	sEcSlaveAmsNetAdr:T_AmsNetId;
	rValue:REAL;
	bOverrange, bDataInvalid, bError, bCalibrationInProgress, bSteadyState:BOOL;
	bTxPDOToggle, bSyncError:BOOL;
	sfFullCalibration:R_TRIG;
	sfZeroCalibration:R_TRIG;
	sfTara:R_TRIG;
	sfTaraEEProm:R_TRIG;
	fbCoE:FB_EcCoESdoWrite;
	wCoeData:WORD;
	sStatus, sSampleMode:STRING(100);
	bTermError:BOOL;
	nCntCalibrations:UDINT;
	sfCalibInProgress:R_TRIG;
	sfLoadReference:R_TRIG;
	sfScaleFactor:R_TRIG;
	rValueDiff, rValueL:REAL;
	bActivateAutoInputFreeze:BOOL;
	rInputFreezeTreshold:REAL:=10;
	tofInputFreeze:TOF;
	tInputFreeze:TIME:=t#50ms;
	sfCntInputFreeze:R_TRIG;
	nCntInputFreeze:UDINT;
	rScaleFactor :REAL:=1.0;
	bCmdScaleFactor:BOOL;


END_VAR

(*EP3356-0022)	para celdas de carga*)
(*toma de datos*)
bOverrange		:= wStatus.1;
bDataInvalid	:= wStatus.3;
bError			:= wStatus.6;
bCalibrationInProgress := wStatus.7;
bSteadyState	:= wStatus.8;
bSyncError		:= wStatus.13;
bTxPDOToggle	:= wStatus.15;

(*triggers*)
sfScaleFactor(CLK:=bCmdScaleFactor);
sfZeroCalibration(CLK:=bCmd_ZeroCalibration);
sfFullCalibration(CLK:=bCmd_FullCalibration);
sfTara(CLK:=bCmd_Tara);
sfTaraEEProm(CLK:=bCmd_TaraEEProm);
sfLoadReference(CLK:=bCmd_LoadReference);

(*value: Integer or Real value*)
IF (rValue_REAL <> 0) THEN	(*select currently used input data*)
	rValue := rValue_REAL;
ELSIF (nValue_DINT <> 0) THEN
	rValue := DINT_TO_REAL(nValue_DINT)/1000;
ELSE
	rValue := 0;
END_IF

(*status*)
IF bWcState THEN
	sStatus := 'Wc fail';
	bTermError := TRUE;
ELSIF NOT (wState.3) THEN
	sStatus := 'Slave not in OP';
	bTermError := TRUE;
ELSIF bDataInvalid THEN
	sStatus := 'DataInvalid';
	bTermError := TRUE;
ELSIF bError THEN
	sStatus := 'Channel Error';
	bTermError := TRUE;
ELSIF bOverrange THEN
	sStatus := 'Overrange';
	bTermError := TRUE;
ELSE
	sStatus := 'ok';
	bTermError := FALSE;
END_IF

	(*sample mode 0/1*)
sSampleMode := SEL(bSampleMode, '0', '1');

	(*count calibrations*)
sfCalibInProgress(CLK:= bCalibrationInProgress, Q=> );
nCntCalibrations := SEL(sfCalibInProgress.Q , nCntCalibrations, nCntCalibrations+ 1);

	(*Coe parameter administration*)
sEcSlaveAmsNetAdr := F_CreateAmsNetId(nIds:=stEcSlaveAmsNetAdr.netId );

	(*test input freeze
this lines are for a small demonstration of Input freeze: when difference of loadvalue, compared to last PLC cycle, is over rInputFreezeTreshold
then InputFreeze is activated by tofInputFreeze for some time. See screenshot in documentation for further explanations*)
rValueDiff := rValue - rValueL;
rValueL := rValue;
tofInputFreeze(IN:= bActivateAutoInputFreeze AND (ABS(rValueDiff) >rInputFreezeTreshold) , PT:= tInputFreeze, Q=> , ET=> );
sfCntInputFreeze(CLK:= tofInputFreeze.Q , Q=> );
nCntInputFreeze := SEL(sfCntInputFreeze.Q , nCntInputFreeze, nCntInputFreeze+ 1);

(*++++++++++++++ comunicacion CoE  ++++++++++++++++++++++*)
(* Scale factor*)
fbCoE(
	sNetId		:= sEcSlaveAmsNetAdr,
	nSlaveAddr 	:= stEcSlaveAmsNetAdr.port,
	nSubIndex 	:= 16#27,
	nIndex 		:= 16#8000,
	pSrcBuf 	:= ADR(rScaleFactor),
	cbBufLen 	:= SIZEOF(rScaleFactor),
	bExecute 	:= sfScaleFactor.Q,
	tTimeout 	:= t#5s
);

wCoeData := 16#0101; (* Comando zerocalibration*)
fbCoE(
	sNetId		:= sEcSlaveAmsNetAdr,
	nSlaveAddr 	:= stEcSlaveAmsNetAdr.port,
	nSubIndex 	:= 16#01,
	nIndex 		:= 16#FB00,
	pSrcBuf 	:= ADR(wCoeData),
	cbBufLen 	:= SIZEOF(wCoeData),
	bExecute 	:= sfZeroCalibration.Q,
	tTimeout 	:= t#5s
);

wCoeData := 16#0102; (* calibracion*)
fbCoE(
	sNetId		:= sEcSlaveAmsNetAdr,
	nSlaveAddr 	:= stEcSlaveAmsNetAdr.port,
	nSubIndex 	:= 16#01,
	nIndex 		:= 16#FB00,
	pSrcBuf 	:= ADR(wCoeData),
	cbBufLen 	:= SIZEOF(wCoeData),
	bExecute 	:= sfFullCalibration.Q,
	tTimeout 	:= t#5s
);

wCoeData := 16#0001; (* tara*)
fbCoE(
	sNetId		:= sEcSlaveAmsNetAdr,
	nSlaveAddr 	:= stEcSlaveAmsNetAdr.port,
	nSubIndex 	:= 16#01,
	nIndex 		:= 16#FB00,
	pSrcBuf 	:= ADR(wCoeData),
	cbBufLen 	:= SIZEOF(wCoeData),
	bExecute 	:= sfTara.Q,
	tTimeout 	:= t#5s
);

wCoeData := 16#0002; (* tara EEProm*)
fbCoE(
	sNetId		:= sEcSlaveAmsNetAdr,
	nSlaveAddr 	:= stEcSlaveAmsNetAdr.port,
	nSubIndex 	:= 16#01,
	nIndex 		:= 16#FB00,
	pSrcBuf 	:= ADR(wCoeData),
	cbBufLen 	:= SIZEOF(wCoeData),
	bExecute 	:= sfTaraEEProm.Q,
	tTimeout 	:= t#5s
);

(* load reference*)
fbCoE(
	sNetId		:= sEcSlaveAmsNetAdr,
	nSlaveAddr 	:= stEcSlaveAmsNetAdr.port,
	nSubIndex 	:= 16#28,
	nIndex 		:= 16#8000,
	pSrcBuf 	:= ADR(fLoadReference),
	cbBufLen 	:= SIZEOF(fLoadReference),
	bExecute 	:= sfLoadReference.Q,
	tTimeout 	:= t#5s
);


	(*output data to terminal*)
wControl.0 := bStartManualCalib;
wControl.1 := bDisableCalibration;
wControl.2 := bInputFreeze OR tofInputFreeze.Q ;
wControl.3 := bSampleMode;
wControl.4 := bTara;

END_FUNCTION_BLOCK

// ---- POUs/Tabla_FIFO.TcPOU
FUNCTION_BLOCK Tabla_FIFO
VAR_INPUT 
	Dato :REAL;
END_VAR
VAR_OUTPUT
END_VAR
VAR_IN_OUT
	Tabla :ARRAY [1..10]OF REAL;
	Trigger :BOOL;
END_VAR
VAR
	posicion: INT;
END_VAR

IF trigger  THEN
	posicion:=1;
	FOR posicion:=10 TO 2 BY -1 DO
	Tabla[posicion]:=Tabla[posicion-1];
	END_FOR;
	Tabla[1]:=Dato;
	trigger:=FALSE;
END_IF

END_FUNCTION_BLOCK

// ---- POUs/Perifericos/Descarga_semilla.TcPOU
PROGRAM Descarga_semilla
VAR
	fbPE_B_VF1 :Equipo_Motor_ATV320;//Elevador embolse
	PE_B1_V1: Equipo_Valvula_5_2_biestable;
	PE_B1_V1_CmdAuto_Pos1:BOOL;
	PE_B1_V1_CmdAuto_Pos2:BOOL;
	PE_B2_V1: Equipo_Valvula_5_2_biestable;
	PE_B2_V1_CmdAuto_Pos1:BOOL;
	PE_B2_V1_CmdAuto_Pos2:BOOL;
	PE_B3_V1: Equipo_Valvula_5_2_biestable;
	PE_B3_V1_CmdAuto_Pos1:BOOL;
	PE_B3_V1_CmdAuto_Pos2:BOOL;
	PE_B1_V2_CmdAuto:BOOL;
	PE_B2_V2_CmdAuto:BOOL;
	PE_B3_V2_CmdAuto:BOOL;	
	
	bHS :BOOL;
	dintHS	:DINT:=3;
	Tmr_B1_LLS: TON;
	B1_LLS_Ok: BOOL;
	Tmr_B2_LLS: TON;
	B2_LLS_Ok: BOOL;
	TmrCicloCarga: TON;
	Cargar_B2: BOOL;
	AuxCargar_B2: BOOL;
	AuxB1_V1: BOOL;
	AuxB2_V1: BOOL;
	TmrDemoraB2_V1: TOF;
	TmrPE_B1_HLS: TON;	//Nível alto da caixa de sacarias
	TmrPE_B2_HLS: TON;	//Nível alto do BIGBAG 2
	TmrPE_B3_HLS: TON;	//Nível alto do BIGBAG 3
	TDemoraPE_B1_LLS: TON;
	TDemoraPE_BE2_LLS: TON;
	TDemoraPE_BE3_LLS: TON;
	Tmr_B3_LLS: TON;
	B3_LLS_Ok: BOOL;
	Tiempo_seg_to_TIME_PE_B_VF1: Tiempo_seg_to_TIME;
	TmrDemoraPE_B_VF1: TOF;
	TDemoraB3_V1: TOF;
	PE_B1_V1_Teste: Equipo_Valvula_5_2;
	PE_B1_V2_Teste: Equipo_Valvula_5_2;
	PE_B1_V3_Teste: Equipo_Valvula_5_2;
	TON_CaixaCheia: TON;
	PausaEnsaque: BOOL;	//Se as duas caixas de ensaque estiverem cheias e a descarga for no bigbag, pausa o processo
	// Atraso na descarga da caixa 3 para que não passem canecas cheias
	TOF_DescargaCX3: TOF;
END_VAR
VAR // added by the converter: edge detectors and wires of the graphical bodies
    _w1 : BOOL;
    _rt1 : R_TRIG;
END_VAR

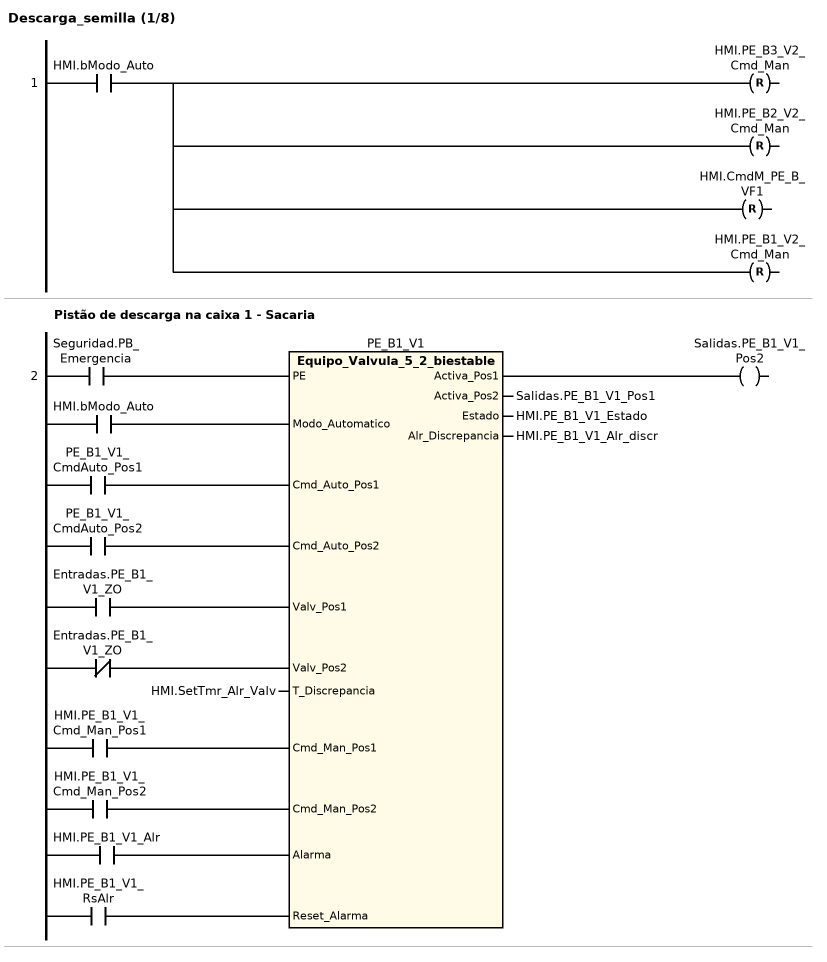
// NETWORK 1
_w1 := HMI.bModo_Auto;
HMI.PE_B3_V2_Cmd_Man R= _w1;
HMI.PE_B2_V2_Cmd_Man R= _w1;
HMI.CmdM_PE_B_VF1 R= _w1;
HMI.PE_B1_V2_Cmd_Man R= _w1;

// NETWORK 2: Pistão de descarga na caixa 1 - Sacaria
PE_B1_V1(
    PE := Seguridad.PB_Emergencia,
    Modo_Automatico := HMI.bModo_Auto,
    Cmd_Auto_Pos1 := PE_B1_V1_CmdAuto_Pos1,
    Cmd_Auto_Pos2 := PE_B1_V1_CmdAuto_Pos2,
    Valv_Pos1 := Entradas.PE_B1_V1_ZO,
    Valv_Pos2 := NOT Entradas.PE_B1_V1_ZO,
    T_Discrepancia := HMI.SetTmr_Alr_Valv,
    Cmd_Man_Pos1 := HMI.PE_B1_V1_Cmd_Man_Pos1,
    Cmd_Man_Pos2 := HMI.PE_B1_V1_Cmd_Man_Pos2,
    Alarma := HMI.PE_B1_V1_Alr,
    Reset_Alarma := HMI.PE_B1_V1_RsAlr,
    Activa_Pos2 => Salidas.PE_B1_V1_Pos1,
    Estado => HMI.PE_B1_V1_Estado,
    Alr_Discrepancia => HMI.PE_B1_V1_Alr_discr); // Equipo_Valvula_5_2_biestable
Salidas.PE_B1_V1_Pos2 := PE_B1_V1.Activa_Pos1;

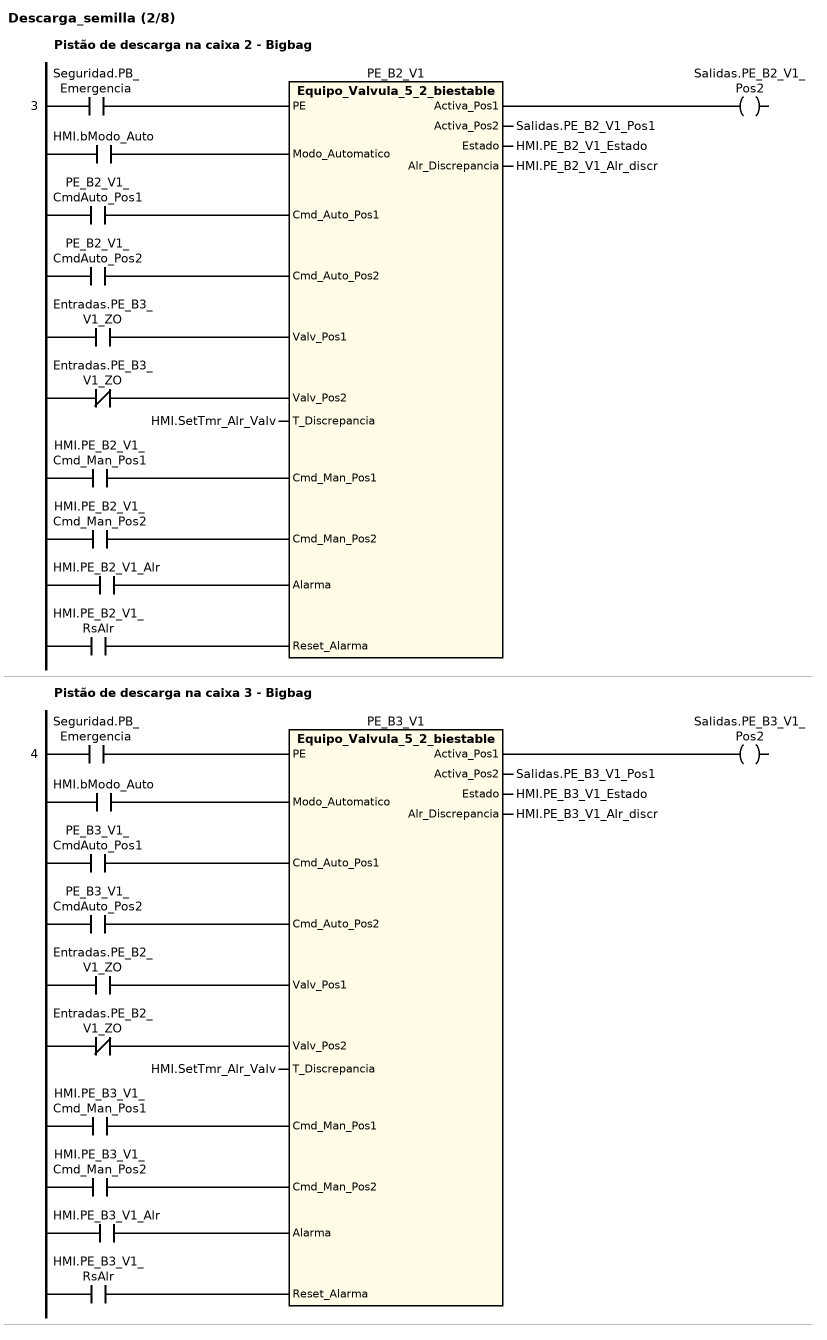
// NETWORK 3: Pistão de descarga na caixa 2 - Bigbag
PE_B2_V1(
    PE := Seguridad.PB_Emergencia,
    Modo_Automatico := HMI.bModo_Auto,
    Cmd_Auto_Pos1 := PE_B2_V1_CmdAuto_Pos1,
    Cmd_Auto_Pos2 := PE_B2_V1_CmdAuto_Pos2,
    Valv_Pos1 := Entradas.PE_B3_V1_ZO,
    Valv_Pos2 := NOT Entradas.PE_B3_V1_ZO,
    T_Discrepancia := HMI.SetTmr_Alr_Valv,
    Cmd_Man_Pos1 := HMI.PE_B2_V1_Cmd_Man_Pos1,
    Cmd_Man_Pos2 := HMI.PE_B2_V1_Cmd_Man_Pos2,
    Alarma := HMI.PE_B2_V1_Alr,
    Reset_Alarma := HMI.PE_B2_V1_RsAlr,
    Activa_Pos2 => Salidas.PE_B2_V1_Pos1,
    Estado => HMI.PE_B2_V1_Estado,
    Alr_Discrepancia => HMI.PE_B2_V1_Alr_discr); // Equipo_Valvula_5_2_biestable
Salidas.PE_B2_V1_Pos2 := PE_B2_V1.Activa_Pos1;

// NETWORK 4: Pistão de descarga na caixa 3 - Bigbag
PE_B3_V1(
    PE := Seguridad.PB_Emergencia,
    Modo_Automatico := HMI.bModo_Auto,
    Cmd_Auto_Pos1 := PE_B3_V1_CmdAuto_Pos1,
    Cmd_Auto_Pos2 := PE_B3_V1_CmdAuto_Pos2,
    Valv_Pos1 := Entradas.PE_B2_V1_ZO,
    Valv_Pos2 := NOT Entradas.PE_B2_V1_ZO,
    T_Discrepancia := HMI.SetTmr_Alr_Valv,
    Cmd_Man_Pos1 := HMI.PE_B3_V1_Cmd_Man_Pos1,
    Cmd_Man_Pos2 := HMI.PE_B3_V1_Cmd_Man_Pos2,
    Alarma := HMI.PE_B3_V1_Alr,
    Reset_Alarma := HMI.PE_B3_V1_RsAlr,
    Activa_Pos2 => Salidas.PE_B3_V1_Pos1,
    Estado => HMI.PE_B3_V1_Estado,
    Alr_Discrepancia => HMI.PE_B3_V1_Alr_discr); // Equipo_Valvula_5_2_biestable
Salidas.PE_B3_V1_Pos2 := PE_B3_V1.Activa_Pos1;

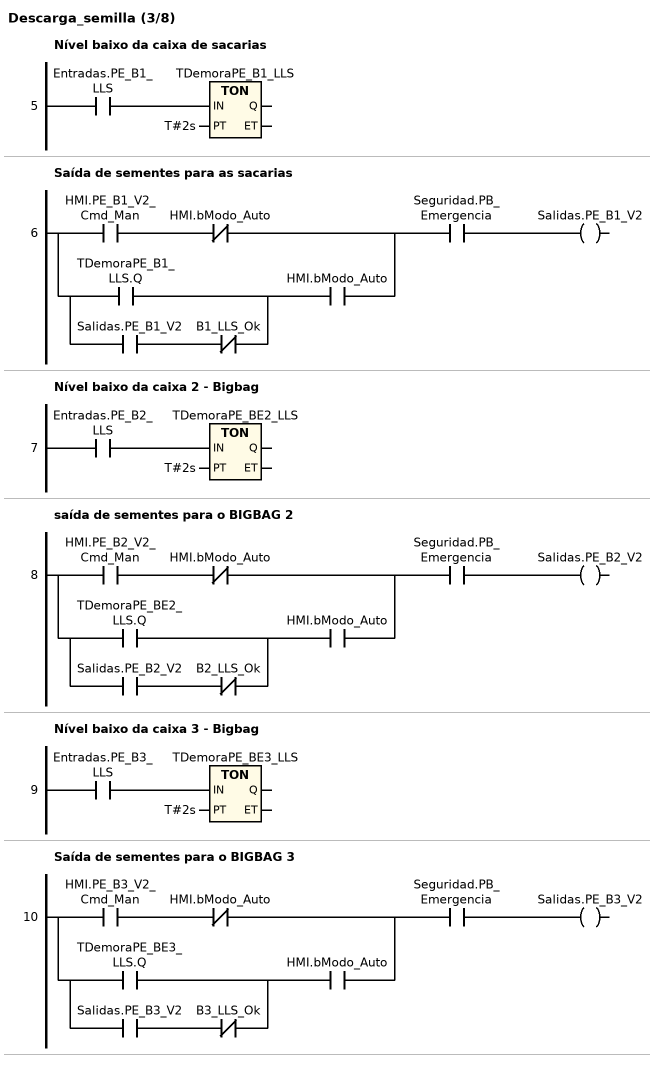
// NETWORK 5: Nível baixo da caixa de sacarias
TDemoraPE_B1_LLS(IN := Entradas.PE_B1_LLS, PT := T#2s); // TON

// NETWORK 6: Saída de sementes para as sacarias
Salidas.PE_B1_V2 := (HMI.PE_B1_V2_Cmd_Man AND NOT HMI.bModo_Auto OR (TDemoraPE_B1_LLS.Q OR Salidas.PE_B1_V2 AND NOT B1_LLS_Ok) AND HMI.bModo_Auto) AND Seguridad.PB_Emergencia;

// NETWORK 7: Nível baixo da caixa 2 - Bigbag
TDemoraPE_BE2_LLS(IN := Entradas.PE_B2_LLS, PT := T#2s); // TON

// NETWORK 8: saída de sementes para o BIGBAG 2
Salidas.PE_B2_V2 := (HMI.PE_B2_V2_Cmd_Man AND NOT HMI.bModo_Auto OR (TDemoraPE_BE2_LLS.Q OR Salidas.PE_B2_V2 AND NOT B2_LLS_Ok) AND HMI.bModo_Auto) AND Seguridad.PB_Emergencia;

// NETWORK 9: Nível baixo da caixa 3 - Bigbag
TDemoraPE_BE3_LLS(IN := Entradas.PE_B3_LLS, PT := T#2s); // TON

// NETWORK 10: Saída de sementes para o BIGBAG 3
Salidas.PE_B3_V2 := (HMI.PE_B3_V2_Cmd_Man AND NOT HMI.bModo_Auto OR (TDemoraPE_BE3_LLS.Q OR Salidas.PE_B3_V2 AND NOT B3_LLS_Ok) AND HMI.bModo_Auto) AND Seguridad.PB_Emergencia;

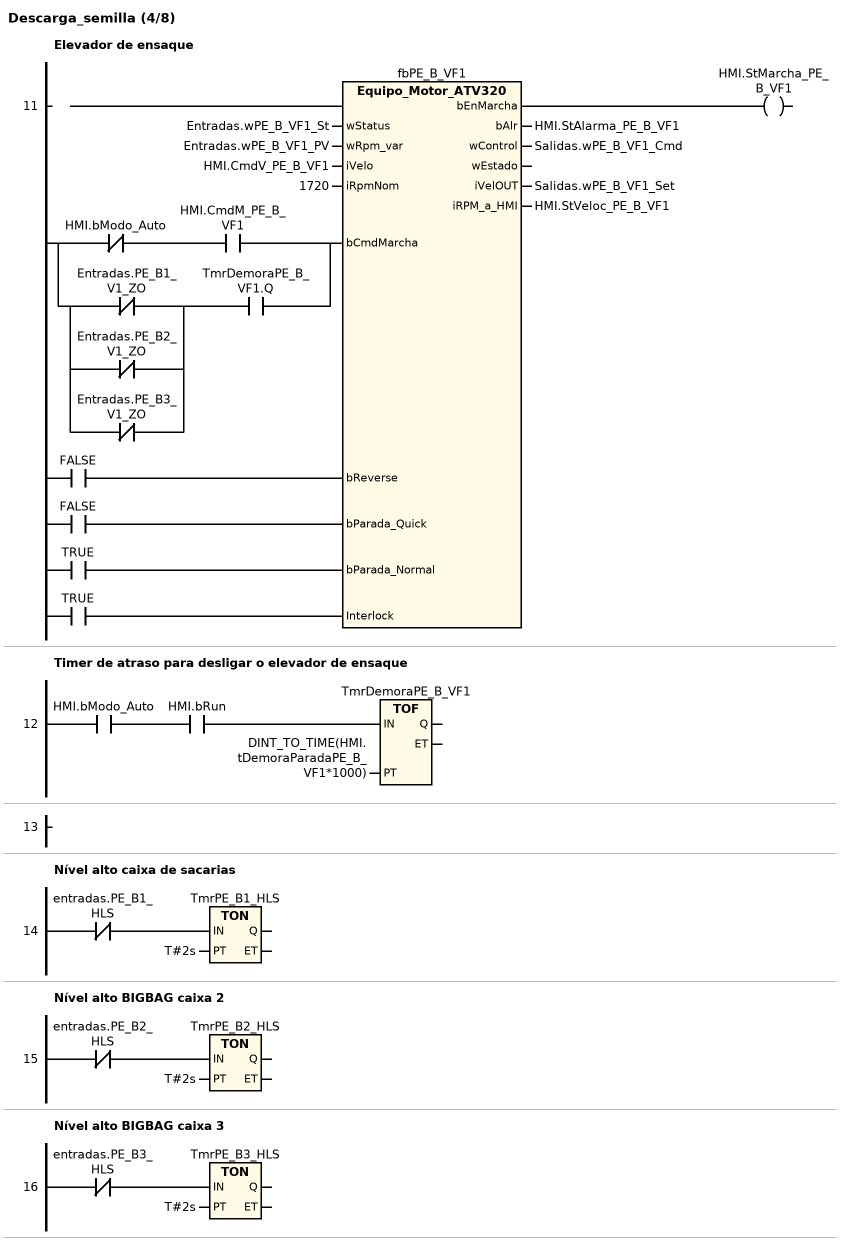
// NETWORK 11: Elevador de ensaque
fbPE_B_VF1(
    wStatus := Entradas.wPE_B_VF1_St,
    wRpm_var := Entradas.wPE_B_VF1_PV,
    iVelo := HMI.CmdV_PE_B_VF1,
    iRpmNom := 1720,
    bCmdMarcha := NOT HMI.bModo_Auto AND HMI.CmdM_PE_B_VF1 OR (NOT Entradas.PE_B1_V1_ZO OR NOT Entradas.PE_B2_V1_ZO OR NOT Entradas.PE_B3_V1_ZO) AND TmrDemoraPE_B_VF1.Q,
    bReverse := FALSE,
    bParada_Quick := FALSE,
    bParada_Normal := TRUE,
    Interlock := TRUE,
    bAlr => HMI.StAlarma_PE_B_VF1,
    wControl => Salidas.wPE_B_VF1_Cmd,
    iVelOUT => Salidas.wPE_B_VF1_Set,
    iRPM_a_HMI => HMI.StVeloc_PE_B_VF1); // Equipo_Motor_ATV320
HMI.StMarcha_PE_B_VF1 := fbPE_B_VF1.bEnMarcha;

// NETWORK 12: Timer de atraso para desligar o elevador de ensaque
TmrDemoraPE_B_VF1(IN := HMI.bModo_Auto AND HMI.bRun, PT := DINT_TO_TIME(HMI.tDemoraParadaPE_B_VF1*1000)); // TOF

// NETWORK 13

// NETWORK 14: Nível alto caixa de sacarias
TmrPE_B1_HLS(IN := NOT entradas.PE_B1_HLS, PT := T#2s); // TON

// NETWORK 15: Nível alto BIGBAG caixa 2
TmrPE_B2_HLS(IN := NOT entradas.PE_B2_HLS, PT := T#2s); // TON

// NETWORK 16: Nível alto BIGBAG caixa 3
TmrPE_B3_HLS(IN := NOT entradas.PE_B3_HLS, PT := T#2s); // TON

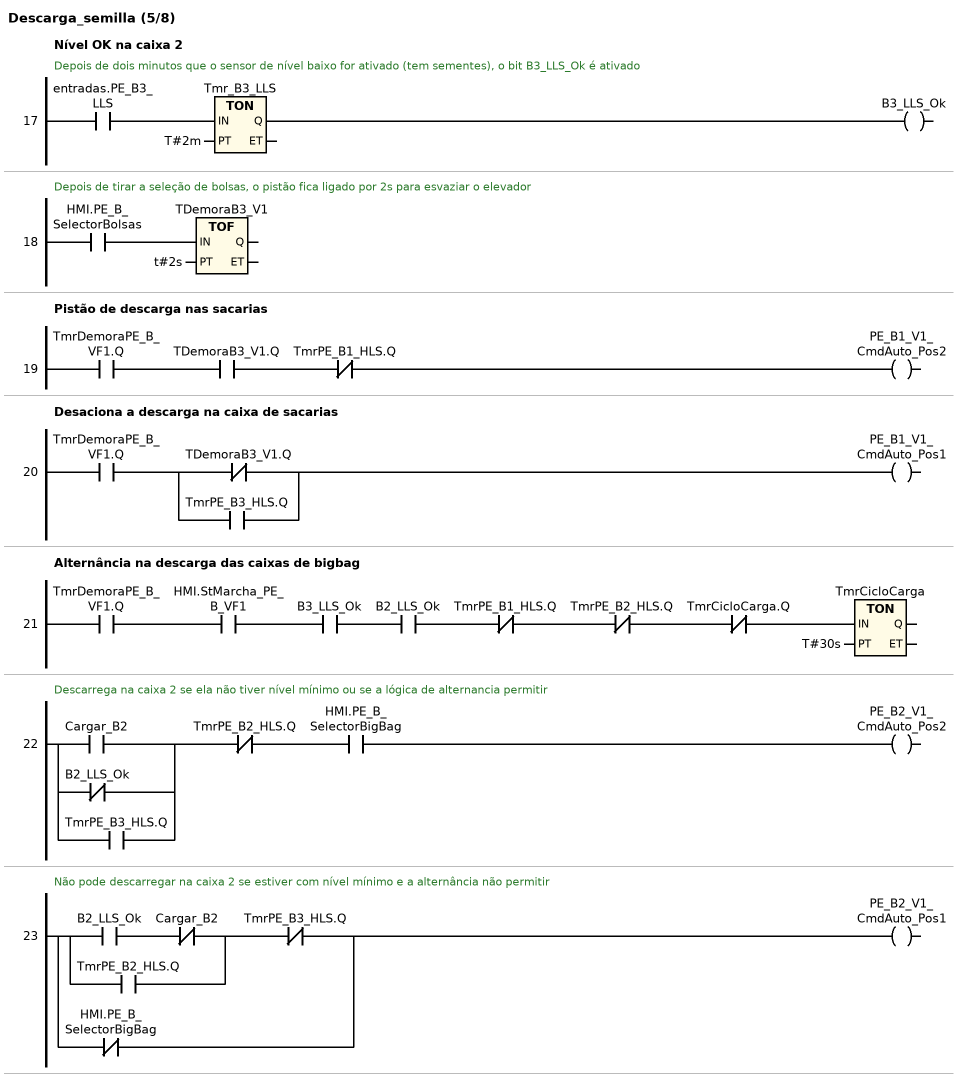
// NETWORK 17: Nível OK na caixa 2
// Depois de dois minutos que o sensor de nível baixo for ativado (tem sementes), o bit B3_LLS_Ok é ativado
Tmr_B3_LLS(IN := entradas.PE_B3_LLS, PT := T#2m); // TON
B3_LLS_Ok := Tmr_B3_LLS.Q;

// NETWORK 18
// Depois de tirar a seleção de bolsas, o pistão fica ligado por 2s para esvaziar o elevador
TDemoraB3_V1(IN := HMI.PE_B_SelectorBolsas, PT := t#2s); // TOF

// NETWORK 19: Pistão de descarga nas sacarias
PE_B1_V1_CmdAuto_Pos2 := TmrDemoraPE_B_VF1.Q AND TDemoraB3_V1.Q AND NOT TmrPE_B1_HLS.Q;

// NETWORK 20: Desaciona a descarga na caixa de sacarias
PE_B1_V1_CmdAuto_Pos1 := TmrDemoraPE_B_VF1.Q AND (NOT TDemoraB3_V1.Q OR TmrPE_B3_HLS.Q);

// NETWORK 21: Alternância na descarga das caixas de bigbag
TmrCicloCarga(IN := TmrDemoraPE_B_VF1.Q AND HMI.StMarcha_PE_B_VF1 AND B3_LLS_Ok AND B2_LLS_Ok AND NOT TmrPE_B1_HLS.Q AND NOT TmrPE_B2_HLS.Q AND NOT TmrCicloCarga.Q, PT := T#30s); // TON

// NETWORK 22
// Descarrega na caixa 2 se ela não tiver nível mínimo ou se a lógica de alternancia permitir
PE_B2_V1_CmdAuto_Pos2 := (Cargar_B2 OR NOT B2_LLS_Ok OR TmrPE_B3_HLS.Q) AND NOT TmrPE_B2_HLS.Q AND HMI.PE_B_SelectorBigBag;

// NETWORK 23
// Não pode descarregar na caixa 2 se estiver com nível mínimo e a alternância não permitir
PE_B2_V1_CmdAuto_Pos1 := (B2_LLS_Ok AND NOT Cargar_B2 OR TmrPE_B2_HLS.Q) AND NOT TmrPE_B3_HLS.Q OR NOT HMI.PE_B_SelectorBigBag;

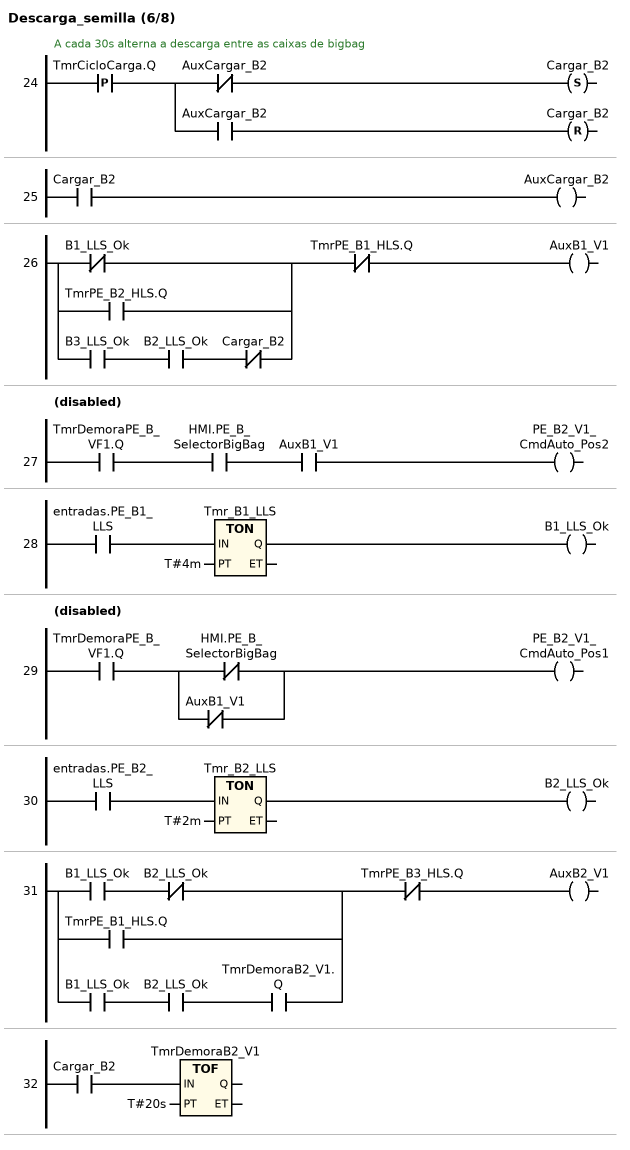
// NETWORK 24
// A cada 30s alterna a descarga entre as caixas de bigbag
_rt1(CLK := TmrCicloCarga.Q);
Cargar_B2 S= _rt1.Q AND NOT AuxCargar_B2;
Cargar_B2 R= _rt1.Q AND AuxCargar_B2;

// NETWORK 25
AuxCargar_B2 := Cargar_B2;

// NETWORK 26
AuxB1_V1 := (NOT B1_LLS_Ok OR TmrPE_B2_HLS.Q OR B3_LLS_Ok AND B2_LLS_Ok AND NOT Cargar_B2) AND NOT TmrPE_B1_HLS.Q;

// NETWORK 27 (disabled)
// PE_B2_V1_CmdAuto_Pos2 := TmrDemoraPE_B_VF1.Q AND HMI.PE_B_SelectorBigBag AND AuxB1_V1;

// NETWORK 28
Tmr_B1_LLS(IN := entradas.PE_B1_LLS, PT := T#4m); // TON
B1_LLS_Ok := Tmr_B1_LLS.Q;

// NETWORK 29 (disabled)
// PE_B2_V1_CmdAuto_Pos1 := TmrDemoraPE_B_VF1.Q AND (NOT HMI.PE_B_SelectorBigBag OR NOT AuxB1_V1);

// NETWORK 30
Tmr_B2_LLS(IN := entradas.PE_B2_LLS, PT := T#2m); // TON
B2_LLS_Ok := Tmr_B2_LLS.Q;

// NETWORK 31
AuxB2_V1 := (B1_LLS_Ok AND NOT B2_LLS_Ok OR TmrPE_B1_HLS.Q OR B1_LLS_Ok AND B2_LLS_Ok AND TmrDemoraB2_V1.Q) AND NOT TmrPE_B3_HLS.Q;

// NETWORK 32
TmrDemoraB2_V1(IN := Cargar_B2, PT := T#20s); // TOF

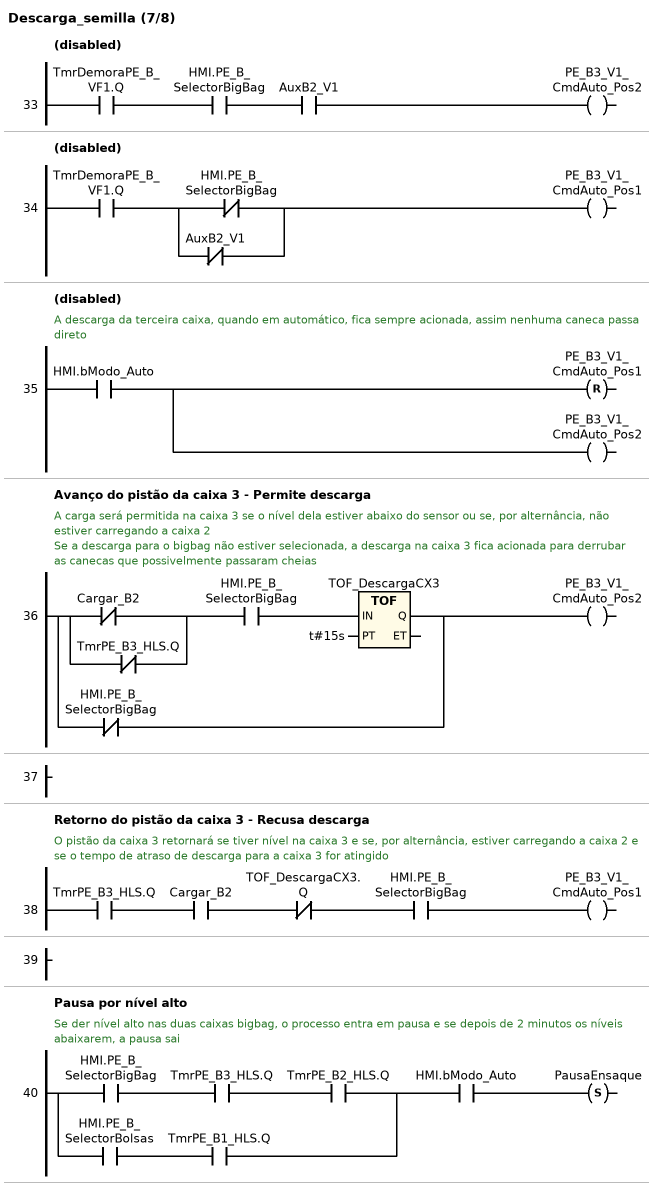
// NETWORK 33 (disabled)
// PE_B3_V1_CmdAuto_Pos2 := TmrDemoraPE_B_VF1.Q AND HMI.PE_B_SelectorBigBag AND AuxB2_V1;

// NETWORK 34 (disabled)
// PE_B3_V1_CmdAuto_Pos1 := TmrDemoraPE_B_VF1.Q AND (NOT HMI.PE_B_SelectorBigBag OR NOT AuxB2_V1);

// NETWORK 35 (disabled)
// A descarga da terceira caixa, quando em automático, fica sempre acionada, assim nenhuma caneca passa direto
// PE_B3_V1_CmdAuto_Pos1 R= HMI.bModo_Auto;
// PE_B3_V1_CmdAuto_Pos2 := HMI.bModo_Auto;

// NETWORK 36: Avanço do pistão da caixa 3 - Permite descarga
// A carga será permitida na caixa 3 se o nível dela estiver abaixo do sensor ou se, por alternância, não estiver carregando a caixa 2
// Se a descarga para o bigbag não estiver selecionada, a descarga na caixa 3 fica acionada para derrubar as canecas que possivelmente passaram cheias
TOF_DescargaCX3(IN := (NOT Cargar_B2 OR NOT TmrPE_B3_HLS.Q) AND HMI.PE_B_SelectorBigBag, PT := t#15s); // TOF
PE_B3_V1_CmdAuto_Pos2 := TOF_DescargaCX3.Q OR NOT HMI.PE_B_SelectorBigBag;

// NETWORK 37

// NETWORK 38: Retorno do pistão da caixa 3 - Recusa descarga
// O pistão da caixa 3 retornará se tiver nível na caixa 3 e se, por alternância, estiver carregando a caixa 2 e se o tempo de atraso de descarga para a caixa 3 for atingido
PE_B3_V1_CmdAuto_Pos1 := TmrPE_B3_HLS.Q AND Cargar_B2 AND NOT TOF_DescargaCX3.Q AND HMI.PE_B_SelectorBigBag;

// NETWORK 39

// NETWORK 40: Pausa por nível alto
// Se der nível alto nas duas caixas bigbag, o processo entra em pausa e se depois de 2 minutos os níveis abaixarem, a pausa sai
PausaEnsaque S= (HMI.PE_B_SelectorBigBag AND TmrPE_B3_HLS.Q AND TmrPE_B2_HLS.Q OR HMI.PE_B_SelectorBolsas AND TmrPE_B1_HLS.Q) AND HMI.bModo_Auto;

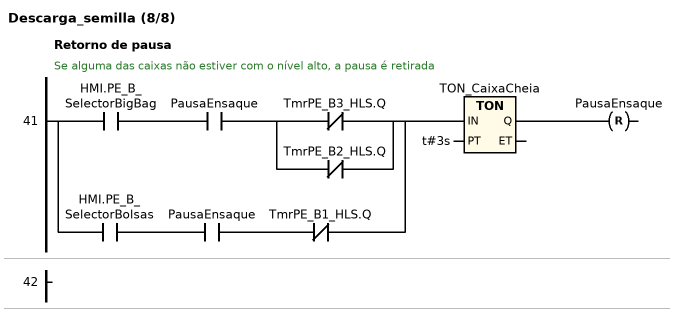
// NETWORK 41: Retorno de pausa
// Se alguma das caixas não estiver com o nível alto, a pausa é retirada
TON_CaixaCheia(IN := HMI.PE_B_SelectorBigBag AND PausaEnsaque AND (NOT TmrPE_B3_HLS.Q OR NOT TmrPE_B2_HLS.Q) OR HMI.PE_B_SelectorBolsas AND PausaEnsaque AND NOT TmrPE_B1_HLS.Q, PT := t#3s); // TON
PausaEnsaque R= TON_CaixaCheia.Q;

// NETWORK 42

END_PROGRAM

// ---- POUs/Control Equipos/Equipo_Valvula_5_2_biestable.TcPOU
FUNCTION_BLOCK Equipo_Valvula_5_2_biestable
VAR_INPUT
	PE				:BOOL; //Parada de emergência
	Modo_Automatico	:BOOL;	//Modo automático
	Cmd_Auto_Pos1	:BOOL;	//Comando para a posição 1
	Cmd_Auto_Pos2	:BOOL;	//Comando para a posição 2
	Valv_Pos1		:BOOL;	//Válvula na posição 1
	Valv_Pos2		:BOOL;	//Válvula na posição 2
	T_Discrepancia	:TIME;	//Tempo para falha na abertura
END_VAR
VAR_OUTPUT
	Activa_Pos1			:BOOL;	//Aciona a saída para a posição 1
	Activa_Pos2			:BOOL;	//Aciona a saída para a posição 2
	Estado				:INT;	//Estado da válvula
	Alr_Discrepancia	:BOOL;	//Em alarme
END_VAR
VAR_IN_OUT
	Cmd_Man_Pos1		:BOOL;	//Comando manual para a posição 1
	Cmd_Man_Pos2		:BOOL;	//Comando manual para a posição 2
	Alarma				:BOOL;	//Em alarme
	Reset_Alarma		:BOOL;	//Reset alarme
END_VAR
VAR_STAT
	FP_Reset			:R_TRIG;	//Borda para reset
	FN_Parada_Auto		:F_TRIG;	//Borda para parada em automático
	FP_Marcha_Auto		:R_TRIG;	//Borda para partir em aitomático
	Cmd_Auto_interno	:BOOL;		//Borda para comando manual
END_VAR

VAR PERSISTENT
	Reset_Eventos		:BOOL;	//Reset contagem de acionamentos
	Timer_Discrepancia		:TON;	//Timer para falha de abertura
	TON_TempoAcionamento	:TON;	//Timer para contar o tempo de acionamento
	R_TRIG_Acionamento		:R_TRIG;	//Borda para tempo de acionamento
	TempoAcionamento		:DINT;	//Tempo de acionamento
	Eventos_Parciales	:DINT;	//Contagem de acionamentos
	Eventos_Totales		:DINT;	//Contagem de eventos totais
END_VAR
VAR // added by the converter: edge detectors and wires of the graphical bodies
    _w1, _w2, _w3, _w4, _w5, _w6, _w7, _w8 : BOOL;
    _rt1, _rt2 : R_TRIG;
END_VAR

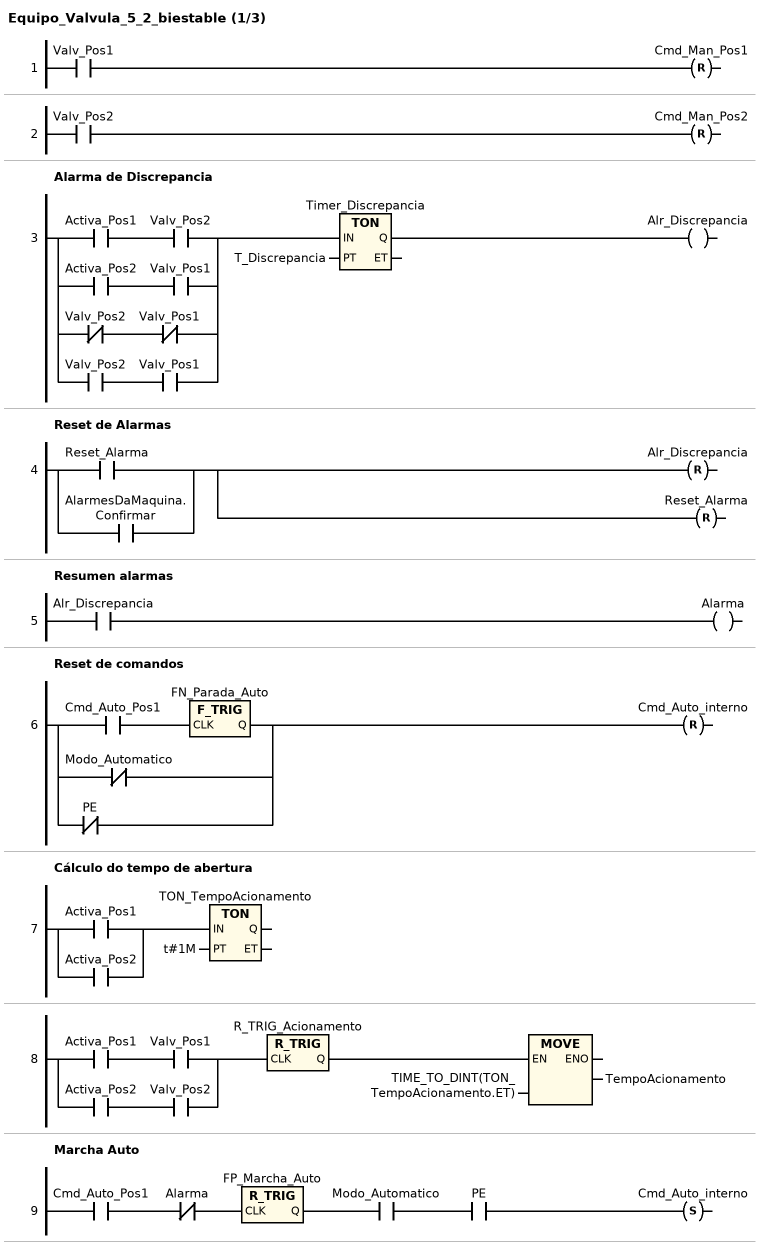
// NETWORK 1
Cmd_Man_Pos1 R= Valv_Pos1;

// NETWORK 2
Cmd_Man_Pos2 R= Valv_Pos2;

// NETWORK 3: Alarma de Discrepancia
Timer_Discrepancia(IN := Activa_Pos1 AND Valv_Pos2 OR Activa_Pos2 AND Valv_Pos1 OR NOT Valv_Pos2 AND NOT Valv_Pos1 OR Valv_Pos2 AND Valv_Pos1, PT := T_Discrepancia); // TON
Alr_Discrepancia := Timer_Discrepancia.Q;

// NETWORK 4: Reset de Alarmas
_w1 := Reset_Alarma OR AlarmesDaMaquina.Confirmar;
Alr_Discrepancia R= _w1;
Reset_Alarma R= _w1;

// NETWORK 5: Resumen alarmas
Alarma := Alr_Discrepancia;

// NETWORK 6: Reset de comandos
FN_Parada_Auto(CLK := Cmd_Auto_Pos1); // F_TRIG
Cmd_Auto_interno R= FN_Parada_Auto.Q OR NOT Modo_Automatico OR NOT PE;

// NETWORK 7: Cálculo do tempo de abertura
TON_TempoAcionamento(IN := Activa_Pos1 OR Activa_Pos2, PT := t#1M); // TON

// NETWORK 8
R_TRIG_Acionamento(CLK := Activa_Pos1 AND Valv_Pos1 OR Activa_Pos2 AND Valv_Pos2); // R_TRIG
IF R_TRIG_Acionamento.Q THEN TempoAcionamento := TIME_TO_DINT(TON_TempoAcionamento.ET); END_IF

// NETWORK 9: Marcha Auto
FP_Marcha_Auto(CLK := Cmd_Auto_Pos1 AND NOT Alarma); // R_TRIG
Cmd_Auto_interno S= FP_Marcha_Auto.Q AND Modo_Automatico AND PE;

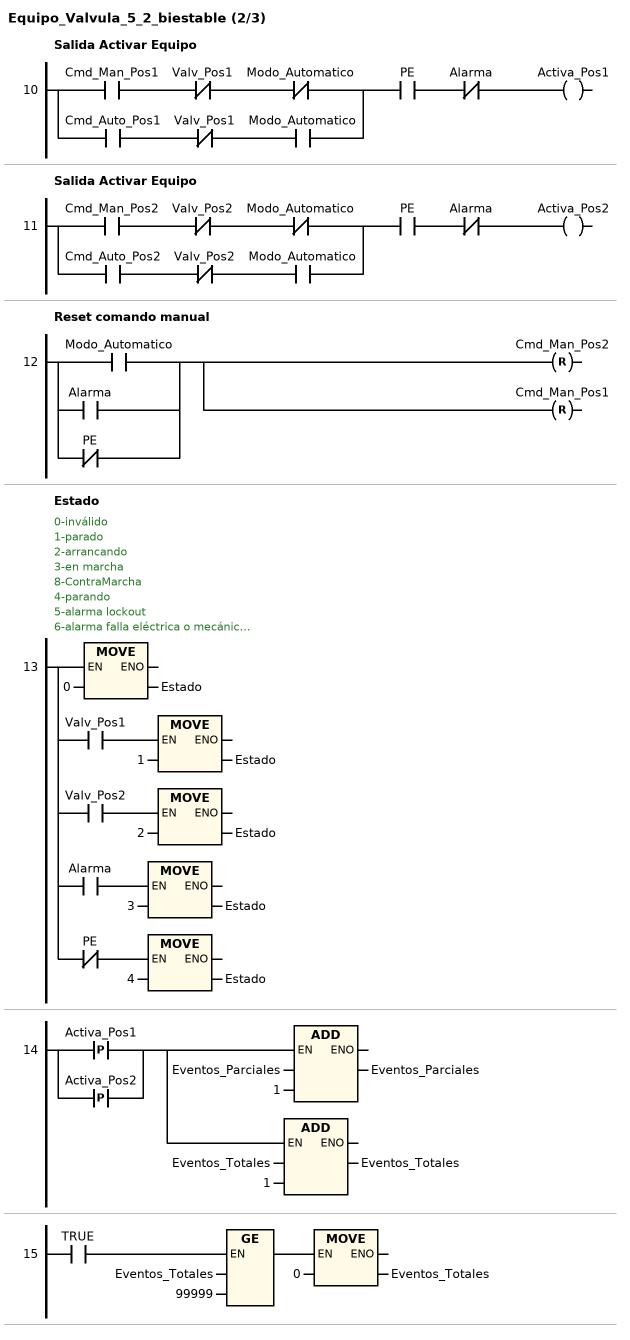
// NETWORK 10: Salida Activar Equipo
Activa_Pos1 := (Cmd_Man_Pos1 AND NOT Valv_Pos1 AND NOT Modo_Automatico OR Cmd_Auto_Pos1 AND NOT Valv_Pos1 AND Modo_Automatico) AND PE AND NOT Alarma;

// NETWORK 11: Salida Activar Equipo
Activa_Pos2 := (Cmd_Man_Pos2 AND NOT Valv_Pos2 AND NOT Modo_Automatico OR Cmd_Auto_Pos2 AND NOT Valv_Pos2 AND Modo_Automatico) AND PE AND NOT Alarma;

// NETWORK 12: Reset comando manual
_w2 := Modo_Automatico OR Alarma OR NOT PE;
Cmd_Man_Pos2 R= _w2;
Cmd_Man_Pos1 R= _w2;

// NETWORK 13: Estado
// 0-inválido
// 1-parado
// 2-arrancando
// 3-en marcha
// 8-ContraMarcha
// 4-parando
// 5-alarma lockout
// 6-alarma falla eléctrica o mecánica
// 7-alarma pulsador emergencia
Estado := 0;
_w3 := Valv_Pos1;
IF _w3 THEN Estado := 1; END_IF
_w4 := Valv_Pos2;
IF _w4 THEN Estado := 2; END_IF
_w5 := Alarma;
IF _w5 THEN Estado := 3; END_IF
_w6 := NOT PE;
IF _w6 THEN Estado := 4; END_IF

// NETWORK 14
_rt1(CLK := Activa_Pos1);
_rt2(CLK := Activa_Pos2);
_w7 := _rt1.Q OR _rt2.Q;
IF _w7 THEN Eventos_Parciales := Eventos_Parciales + 1; END_IF
IF _w7 THEN Eventos_Totales := Eventos_Totales + 1; END_IF

// NETWORK 15
IF Eventos_Totales >= 99999 THEN Eventos_Totales := 0; END_IF

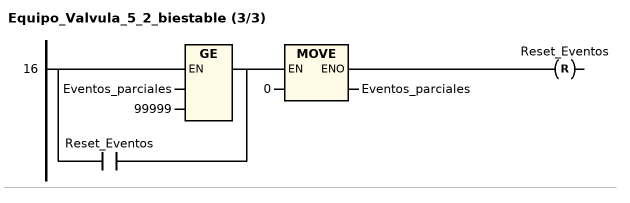
// NETWORK 16
_w8 := Reset_Eventos;
IF NOT _w8 THEN
    _w8 := Eventos_parciales >= 99999;
END_IF
IF _w8 THEN Eventos_parciales := 0; END_IF
Reset_Eventos R= _w8;

END_FUNCTION_BLOCK

// ---- POUs/Testes Thiago/AlarmesDaMaquina.TcPOU
PROGRAM AlarmesDaMaquina
VAR_INPUT
	Confirmar:BOOL;
END_VAR
VAR
	RangeMinimo:REAL := 40;	//Range de abertura mínimo para que as válvulas gerem falha. Em %
	FaltaDeAr	:GeraAlarme;
	Emerg		:GeraAlarme;
	AlrLL		:BOOL;		// Alarme de nível baixo de óleo nas bombas. Se estiver em falso, alguma bomba está com nível baixo
	
	FalhaBomba		:ARRAY[1..12] OF GeraAlarme;	//Bombas de dosagem
	Agitadores		:ARRAY[1..12] OF GeraAlarme;	//Agitadores
	IntervCalibracao:ARRAY[1..12] OF GeraAlarme;	//Tempo de calibração excedido
	IntervLavagem	:ARRAY[1..12] OF GeraAlarme;	//Tempo de lavagem excedido
	NivelOleo		:ARRAY[1..12] OF GeraAlarme;	//nível baixo de óleo
	AnguloValv		:ARRAY[1..48] OF GeraAlarme;	//Falha no angulo de abertura das válvulas
	FalhaValv		:ARRAY[1..48] OF GeraAlarme;	//Falha nas válvulas
	iPC_Diag		:ARRAY[1..5] OF GeraAlarme;		//Alarmes de diagnóstico do iPC
	NivelProd		:ARRAY[1..14] OF GeraAlarme;	//Baixo nível de liquidos e pós
	
	//Elevadores
	FalhaElev1: GeraAlarme;
	FalhaElev2: GeraAlarme;
	FalhaElev3: GeraAlarme;
	
	
	//Dosadores de pó
	FalhaDosador1: GeraAlarme;
	FalhaDosador2: GeraAlarme;
	
	//Homgeneizador e aspersor
	Aspersor: GeraAlarme;
	Homogeneizador: GeraAlarme;

END_VAR

FaltaDeAr(evtEntry:= TC_Events.B300_EventClass.PressaoDeAr, bEvt:= NOT entradas.TR_S_PDI, bConfirm:= Confirmar);	//Baixa pressão de ar
Emerg(evtEntry:= TC_Events.B300_EventClass.Emergencia, bEvt:= NOT Seguridad.PB_Emergencia, bConfirm:= Confirmar);

{Region "Bombas"}
	//Bombas
	FalhaBomba[1](evtEntry	:= TC_Events.B300_EventClass.FalhaBombaLinha1,	bEvt:= Circuito_L1.fbBomba_L1.bAlr, bConfirm:= Confirmar);
	FalhaBomba[2](evtEntry	:= TC_Events.B300_EventClass.FalhaBombaLinha2,	bEvt:= Circuito_L2.fbBomba_L2.bAlr, bConfirm:= Confirmar);
	FalhaBomba[3](evtEntry	:= TC_Events.B300_EventClass.FalhaBombaLinha3,	bEvt:= Circuito_L3.fbBomba_L3.bAlr, bConfirm:= Confirmar);
	FalhaBomba[4](evtEntry	:= TC_Events.B300_EventClass.FalhaBombaLinha4,	bEvt:= Circuito_L4.fbBomba_L4.bAlr, bConfirm:= Confirmar);
	FalhaBomba[5](evtEntry	:= TC_Events.B300_EventClass.FalhaBombaLinha5,	bEvt:= Circuito_L5.fbBomba_L5.bAlr, bConfirm:= Confirmar);
	FalhaBomba[6](evtEntry	:= TC_Events.B300_EventClass.FalhaBombaLinha6,	bEvt:= Circuito_L6.fbBomba_L6.bAlr, bConfirm:= Confirmar);
	FalhaBomba[7](evtEntry	:= TC_Events.B300_EventClass.FalhaBombaLinha7,	bEvt:= Circuito_L7.fbBomba_L7.bAlr, bConfirm:= Confirmar);
	FalhaBomba[8](evtEntry	:= TC_Events.B300_EventClass.FalhaBombaLinha8,	bEvt:= Circuito_L8.fbBomba_L8.bAlr, bConfirm:= Confirmar);
	FalhaBomba[9](evtEntry	:= TC_Events.B300_EventClass.FalhaBombaLinha9,	bEvt:= Circuito_L9.fbBomba_L9.bAlr, bConfirm:= Confirmar);
	FalhaBomba[10](evtEntry	:= TC_Events.B300_EventClass.FalhaBombaLinha10,	bEvt:= Circuito_L10.fbBomba_L10.bAlr, bConfirm:= Confirmar);
	FalhaBomba[11](evtEntry	:= TC_Events.B300_EventClass.FalhaBombaLinha11, bEvt:= Circuito_L11.fbBomba_L11.bAlr, bConfirm:= Confirmar);
	FalhaBomba[12](evtEntry	:= TC_Events.B300_EventClass.FalhaBombaLinha12, bEvt:= Circuito_L12.fbBomba_L12.bAlr, bConfirm:= Confirmar);
	
	//Elevadores
	FalhaElev1(evtEntry:= TC_Events.B300_EventClass.FalhaElevador1, bEvt:= Carga_semilla.fbPE_H_VF1.bAlr, bConfirm:= Confirmar);
	FalhaElev2(evtEntry:= TC_Events.B300_EventClass.FalhaElevador2, bEvt:= Carga_semilla.fbPE_H_VF2.bAlr, bConfirm:= Confirmar);
	FalhaElev3(evtEntry:= TC_Events.B300_EventClass.FalhaElevador3, bEvt:= Descarga_semilla.fbPE_B_VF1.bAlr, bConfirm:= Confirmar);
	
	//Dosadores de pó
	FalhaDosador1(evtEntry:= TC_Events.B300_EventClass.Dosador1, bEvt:= Dosificador_Polvo_1.fbDosificador_P1.bAlr, bConfirm:= Confirmar);
	FalhaDosador2(evtEntry:= TC_Events.B300_EventClass.Dosador2, bEvt:= Dosificador_Polvo_2.fbDosificador_P2.bAlr, bConfirm:= Confirmar);
	
	//Aspersor e homogeneizador
	Aspersor(evtEntry:= TC_Events.B300_EventClass.Aspersor, bEvt:= Tratadora.fbAspersor.bAlr, bConfirm:= Confirmar);
	Homogeneizador(evtEntry:= TC_Events.B300_EventClass.Homogeinizador, bEvt:= Tratadora.fbHomogenizador.bAlr, bConfirm:= Confirmar);
{endregion}

{Region "Nível baixo nas bombas"}
	AlrLL :=	Entradas.bPP1_L1_BD_MangRota AND Entradas.bPP1_L2_BD_MangRota AND Entradas.bPP1_L3_BD_MangRota AND
				Entradas.bPP1_L4_BD_MangRota AND Entradas.bPP2_L5_BD_MangRota AND Entradas.bPP2_L6_BD_MangRota AND
				Entradas.bPP2_L7_BD_MangRota AND Entradas.bPP2_L8_BD_MangRota AND Entradas.bPP3_L9_BD_MangRota AND
				Entradas.bPP3_L10_BD_MangRota AND Entradas.bPP3_L11_BD_MangRota AND Entradas.bPP3_L12_BD_MangRota;
				
	NivelOleo[1](evtEntry:= TC_Events.NivelOleo.BB01, bEvt:= NOT Entradas.bPP1_L1_BD_MangRota, bConfirm:= Confirmar);
	NivelOleo[2](evtEntry:= TC_Events.NivelOleo.BB02, bEvt:= NOT Entradas.bPP1_L2_BD_MangRota, bConfirm:= Confirmar);
	NivelOleo[3](evtEntry:= TC_Events.NivelOleo.BB03, bEvt:= NOT Entradas.bPP1_L3_BD_MangRota, bConfirm:= Confirmar);
	NivelOleo[4](evtEntry:= TC_Events.NivelOleo.BB04, bEvt:= NOT Entradas.bPP1_L4_BD_MangRota, bConfirm:= Confirmar);
	NivelOleo[5](evtEntry:= TC_Events.NivelOleo.BB05, bEvt:= NOT Entradas.bPP2_L5_BD_MangRota, bConfirm:= Confirmar);
	NivelOleo[6](evtEntry:= TC_Events.NivelOleo.BB06, bEvt:= NOT Entradas.bPP2_L6_BD_MangRota, bConfirm:= Confirmar);
	NivelOleo[7](evtEntry:= TC_Events.NivelOleo.BB07, bEvt:= NOT Entradas.bPP2_L7_BD_MangRota, bConfirm:= Confirmar);
	NivelOleo[8](evtEntry:= TC_Events.NivelOleo.BB08, bEvt:= NOT Entradas.bPP2_L8_BD_MangRota, bConfirm:= Confirmar);
	NivelOleo[9](evtEntry:= TC_Events.NivelOleo.BB09, bEvt:= NOT Entradas.bPP3_L9_BD_MangRota, bConfirm:= Confirmar);
	NivelOleo[10](evtEntry:= TC_Events.NivelOleo.BB10, bEvt:= NOT Entradas.bPP3_L10_BD_MangRota, bConfirm:= Confirmar);
	NivelOleo[11](evtEntry:= TC_Events.NivelOleo.BB11, bEvt:= NOT Entradas.bPP3_L11_BD_MangRota, bConfirm:= Confirmar);
	NivelOleo[12](evtEntry:= TC_Events.NivelOleo.BB12, bEvt:= NOT Entradas.bPP3_L12_BD_MangRota, bConfirm:= Confirmar);
{endregion}


{Region "Válvulas"}
	//Válvulas
	//Linha 01
	FalhaValv[1](evtEntry:= TC_Events.Valvulas.Linha1_Valv1, bEvt:= Circuito_L1.Falla_L1_V1, bConfirm:= Confirmar OR HMI.CA1_L1_V1_RsAlr);
	FalhaValv[2](evtEntry:= TC_Events.Valvulas.Linha1_Valv2, bEvt:= Circuito_L1.Falla_L1_V2, bConfirm:= Confirmar OR HMI.CA1_L1_V2_RsAlr);
	FalhaValv[3](evtEntry:= TC_Events.Valvulas.Linha1_Valv3, bEvt:= Circuito_L1.Falla_L1_V3, bConfirm:= Confirmar OR HMI.CA1_L1_V3_RsAlr);
	FalhaValv[4](evtEntry:= TC_Events.Valvulas.Linha1_Valv4, bEvt:= Circuito_L1.Falla_L1_V4, bConfirm:= Confirmar OR HMI.CA1_L1_V4_RsAlr);
	//Linha 02
	FalhaValv[5](evtEntry:= TC_Events.Valvulas.Linha2_Valv1, bEvt:= Circuito_L2.Falla_L2_V1, bConfirm:= Confirmar OR HMI.CA1_L2_V1_RsAlr);
	FalhaValv[6](evtEntry:= TC_Events.Valvulas.Linha2_Valv2, bEvt:= Circuito_L2.Falla_L2_V2, bConfirm:= Confirmar OR HMI.CA1_L2_V2_RsAlr);
	FalhaValv[7](evtEntry:= TC_Events.Valvulas.Linha2_Valv3, bEvt:= Circuito_L2.Falla_L2_V3, bConfirm:= Confirmar OR HMI.CA1_L2_V3_RsAlr);
	FalhaValv[8](evtEntry:= TC_Events.Valvulas.Linha2_Valv4, bEvt:= Circuito_L2.Falla_L2_V4, bConfirm:= Confirmar OR HMI.CA1_L2_V4_RsAlr);
	//Linha 03
	FalhaValv[9](evtEntry:= TC_Events.Valvulas.Linha3_Valv1, bEvt:= Circuito_L3.Falla_L3_V1, bConfirm:= Confirmar OR HMI.CA1_L3_V1_RsAlr);
	FalhaValv[10](evtEntry:= TC_Events.Valvulas.Linha3_Valv2, bEvt:= Circuito_L3.Falla_L3_V2, bConfirm:= Confirmar OR HMI.CA1_L3_V2_RsAlr);
	FalhaValv[11](evtEntry:= TC_Events.Valvulas.Linha3_Valv3, bEvt:= Circuito_L3.Falla_L3_V3, bConfirm:= Confirmar OR HMI.CA1_L3_V3_RsAlr);
	FalhaValv[12](evtEntry:= TC_Events.Valvulas.Linha3_Valv4, bEvt:= Circuito_L3.Falla_L3_V4, bConfirm:= Confirmar OR HMI.CA1_L3_V4_RsAlr);
	//Linha 04
	FalhaValv[13](evtEntry:= TC_Events.Valvulas.Linha4_Valv1, bEvt:= Circuito_L4.Falla_L4_V1, bConfirm:= Confirmar OR HMI.CA1_L4_V1_RsAlr);
	FalhaValv[14](evtEntry:= TC_Events.Valvulas.Linha4_Valv2, bEvt:= Circuito_L4.Falla_L4_V2, bConfirm:= Confirmar OR HMI.CA1_L4_V2_RsAlr);
	FalhaValv[15](evtEntry:= TC_Events.Valvulas.Linha4_Valv3, bEvt:= Circuito_L4.Falla_L4_V3, bConfirm:= Confirmar OR HMI.CA1_L4_V3_RsAlr);
	FalhaValv[16](evtEntry:= TC_Events.Valvulas.Linha4_Valv4, bEvt:= Circuito_L4.Falla_L4_V4, bConfirm:= Confirmar OR HMI.CA1_L4_V4_RsAlr);
	//Linha 05
	FalhaValv[17](evtEntry:= TC_Events.Valvulas.Linha5_Valv1, bEvt:= Circuito_L5.Falla_L5_V1, bConfirm:= Confirmar OR HMI.CA2_L5_V1_RsAlr);
	FalhaValv[18](evtEntry:= TC_Events.Valvulas.Linha5_Valv2, bEvt:= Circuito_L5.Falla_L5_V2, bConfirm:= Confirmar OR HMI.CA2_L5_V2_RsAlr);
	FalhaValv[19](evtEntry:= TC_Events.Valvulas.Linha5_Valv3, bEvt:= Circuito_L5.Falla_L5_V3, bConfirm:= Confirmar OR HMI.CA2_L5_V3_RsAlr);
	FalhaValv[20](evtEntry:= TC_Events.Valvulas.Linha5_Valv4, bEvt:= Circuito_L5.Falla_L5_V4, bConfirm:= Confirmar OR HMI.CA2_L5_V4_RsAlr);
	//Linha 06
	FalhaValv[21](evtEntry:= TC_Events.Valvulas.Linha6_Valv1, bEvt:= Circuito_L6.Falla_L6_V1, bConfirm:= Confirmar OR HMI.CA2_L6_V1_RsAlr);
	FalhaValv[22](evtEntry:= TC_Events.Valvulas.Linha6_Valv2, bEvt:= Circuito_L6.Falla_L6_V2, bConfirm:= Confirmar OR HMI.CA2_L6_V2_RsAlr);
	FalhaValv[23](evtEntry:= TC_Events.Valvulas.Linha6_Valv3, bEvt:= Circuito_L6.Falla_L6_V3, bConfirm:= Confirmar OR HMI.CA2_L6_V3_RsAlr);
	FalhaValv[24](evtEntry:= TC_Events.Valvulas.Linha6_Valv4, bEvt:= Circuito_L6.Falla_L6_V4, bConfirm:= Confirmar OR HMI.CA2_L6_V4_RsAlr);
	//Linha 07
	FalhaValv[25](evtEntry:= TC_Events.Valvulas.Linha7_Valv1, bEvt:= Circuito_L7.Falla_L7_V1, bConfirm:= Confirmar OR HMI.CA2_L7_V1_RsAlr);
	FalhaValv[26](evtEntry:= TC_Events.Valvulas.Linha7_Valv2, bEvt:= Circuito_L7.Falla_L7_V2, bConfirm:= Confirmar OR HMI.CA2_L7_V2_RsAlr);
	FalhaValv[27](evtEntry:= TC_Events.Valvulas.Linha7_Valv3, bEvt:= Circuito_L7.Falla_L7_V3, bConfirm:= Confirmar OR HMI.CA2_L7_V3_RsAlr);
	FalhaValv[28](evtEntry:= TC_Events.Valvulas.Linha7_Valv4, bEvt:= Circuito_L7.Falla_L7_V4, bConfirm:= Confirmar OR HMI.CA2_L7_V4_RsAlr);
	//Linha 08
	FalhaValv[29](evtEntry:= TC_Events.Valvulas.Linha8_Valv1, bEvt:= Circuito_L8.Falla_L8_V1, bConfirm:= Confirmar OR HMI.CA2_L8_V1_RsAlr);
	FalhaValv[30](evtEntry:= TC_Events.Valvulas.Linha8_Valv2, bEvt:= Circuito_L8.Falla_L8_V2, bConfirm:= Confirmar OR HMI.CA2_L8_V2_RsAlr);
	FalhaValv[31](evtEntry:= TC_Events.Valvulas.Linha8_Valv3, bEvt:= Circuito_L8.Falla_L8_V3, bConfirm:= Confirmar OR HMI.CA2_L8_V3_RsAlr);
	FalhaValv[32](evtEntry:= TC_Events.Valvulas.Linha8_Valv4, bEvt:= Circuito_L8.Falla_L8_V4, bConfirm:= Confirmar OR HMI.CA2_L8_V4_RsAlr);
	//Linha 09
	FalhaValv[33](evtEntry:= TC_Events.Valvulas.Linha9_Valv1, bEvt:= Circuito_L9.Falla_L9_V1, bConfirm:= Confirmar OR HMI.CA3_L9_V1_RsAlr);
	FalhaValv[34](evtEntry:= TC_Events.Valvulas.Linha9_Valv2, bEvt:= Circuito_L9.Falla_L9_V2, bConfirm:= Confirmar OR HMI.CA3_L9_V2_RsAlr);
	FalhaValv[35](evtEntry:= TC_Events.Valvulas.Linha9_Valv3, bEvt:= Circuito_L9.Falla_L9_V3, bConfirm:= Confirmar OR HMI.CA3_L9_V3_RsAlr);
	FalhaValv[36](evtEntry:= TC_Events.Valvulas.Linha9_Valv4, bEvt:= Circuito_L9.Falla_L9_V4, bConfirm:= Confirmar OR HMI.CA3_L9_V4_RsAlr);
	//Linha 10
	FalhaValv[37](evtEntry:= TC_Events.Valvulas.Linha10_Valv1, bEvt:= Circuito_L10.Falla_L10_V1, bConfirm:= Confirmar OR HMI.CA3_L10_V1_RsAlr);
	FalhaValv[38](evtEntry:= TC_Events.Valvulas.Linha10_Valv2, bEvt:= Circuito_L10.Falla_L10_V2, bConfirm:= Confirmar OR HMI.CA3_L10_V2_RsAlr);
	FalhaValv[39](evtEntry:= TC_Events.Valvulas.Linha10_Valv3, bEvt:= Circuito_L10.Falla_L10_V3, bConfirm:= Confirmar OR HMI.CA3_L10_V3_RsAlr);
	FalhaValv[40](evtEntry:= TC_Events.Valvulas.Linha10_Valv4, bEvt:= Circuito_L10.Falla_L10_V4, bConfirm:= Confirmar OR HMI.CA3_L10_V4_RsAlr);
	//Linha 11
	FalhaValv[41](evtEntry:= TC_Events.Valvulas.Linha11_Valv1, bEvt:= Circuito_L11.Falla_L11_V1, bConfirm:= Confirmar OR HMI.CA3_L11_V1_RsAlr);
	FalhaValv[42](evtEntry:= TC_Events.Valvulas.Linha11_Valv2, bEvt:= Circuito_L11.Falla_L11_V2, bConfirm:= Confirmar OR HMI.CA3_L11_V2_RsAlr);
	FalhaValv[43](evtEntry:= TC_Events.Valvulas.Linha11_Valv3, bEvt:= Circuito_L11.Falla_L11_V3, bConfirm:= Confirmar OR HMI.CA3_L11_V3_RsAlr);
	FalhaValv[44](evtEntry:= TC_Events.Valvulas.Linha11_Valv4, bEvt:= Circuito_L11.Falla_L11_V4, bConfirm:= Confirmar OR HMI.CA3_L11_V4_RsAlr);
	//Linha 12
	FalhaValv[45](evtEntry:= TC_Events.Valvulas.Linha12_Valv1, bEvt:= Circuito_L12.Falla_L12_V1, bConfirm:= Confirmar OR HMI.CA3_L12_V1_RsAlr);
	FalhaValv[46](evtEntry:= TC_Events.Valvulas.Linha12_Valv2, bEvt:= Circuito_L12.Falla_L12_V2, bConfirm:= Confirmar OR HMI.CA3_L12_V2_RsAlr);
	FalhaValv[47](evtEntry:= TC_Events.Valvulas.Linha12_Valv3, bEvt:= Circuito_L12.Falla_L12_V3, bConfirm:= Confirmar OR HMI.CA3_L12_V3_RsAlr);
	FalhaValv[48](evtEntry:= TC_Events.Valvulas.Linha12_Valv4, bEvt:= Circuito_L12.Falla_L12_V4, bConfirm:= Confirmar OR HMI.CA3_L12_V4_RsAlr);

{endregion}

{Region "Agitadores"}
	//Agitadores
	Agitadores[1](evtEntry:= TC_Events.Agitadores.AgitadorL1, bEvt:= HMI.PP1_L1_AG_Alr, bConfirm:= Confirmar OR HMI.bPP1_L1_AG_RstALr);
	Agitadores[2](evtEntry:= TC_Events.Agitadores.AgitadorL2, bEvt:= HMI.PP1_L2_AG_Alr, bConfirm:= Confirmar OR HMI.bPP1_L2_AG_RstALr);
	Agitadores[3](evtEntry:= TC_Events.Agitadores.AgitadorL3, bEvt:= HMI.PP1_L3_AG_Alr, bConfirm:= Confirmar OR HMI.bPP1_L3_AG_RstALr);
	Agitadores[4](evtEntry:= TC_Events.Agitadores.AgitadorL4, bEvt:= HMI.PP1_L4_AG_Alr, bConfirm:= Confirmar OR HMI.bPP1_L4_AG_RstALr);
	Agitadores[5](evtEntry:= TC_Events.Agitadores.AgitadorL5, bEvt:= HMI.PP2_L5_AG_Alr, bConfirm:= Confirmar OR HMI.bPP2_L5_AG_RstALr);
	Agitadores[6](evtEntry:= TC_Events.Agitadores.AgitadorL6, bEvt:= HMI.PP2_L6_AG_Alr, bConfirm:= Confirmar OR HMI.bPP2_L6_AG_RstALr);
	Agitadores[7](evtEntry:= TC_Events.Agitadores.AgitadorL7, bEvt:= HMI.PP2_L7_AG_Alr, bConfirm:= Confirmar OR HMI.bPP2_L7_AG_RstALr);
	Agitadores[8](evtEntry:= TC_Events.Agitadores.AgitadorL8, bEvt:= HMI.PP2_L8_AG_Alr, bConfirm:= Confirmar OR HMI.bPP2_L8_AG_RstALr);
	Agitadores[9](evtEntry:= TC_Events.Agitadores.AgitadorL9, bEvt:= HMI.PP3_L9_AG_Alr, bConfirm:= Confirmar OR HMI.bPP3_L9_AG_RstALr);
	Agitadores[10](evtEntry:= TC_Events.Agitadores.AgitadorL10, bEvt:= HMI.PP3_L10_AG_Alr, bConfirm:= Confirmar OR HMI.bPP3_L10_AG_RstALr);
	Agitadores[11](evtEntry:= TC_Events.Agitadores.AgitadorL11, bEvt:= HMI.PP3_L11_AG_Alr, bConfirm:= Confirmar OR HMI.bPP3_L11_AG_RstALr);
	Agitadores[12](evtEntry:= TC_Events.Agitadores.AgitadorL12, bEvt:= HMI.PP3_L12_AG_Alr, bConfirm:= Confirmar OR HMI.bPP3_L12_AG_RstALr);
	

{endregion}

{Region "Intervalo de calibração excedido"}
	IntervCalibracao[1](evtEntry:= TC_Events.IntervaloExcedidoCalibracao.Calibracao_L1, bEvt:= DT_TO_UDINT(Main.HoraAtual) - HMI.UltimoAlrCalibr[1] > IntervaloLavCalibr.IntervaloCalibracao * 3600, bConfirm:= Confirmar);
	IntervCalibracao[2](evtEntry:= TC_Events.IntervaloExcedidoCalibracao.Calibracao_L2, bEvt:= DT_TO_UDINT(Main.HoraAtual) - HMI.UltimoAlrCalibr[2] > IntervaloLavCalibr.IntervaloCalibracao * 3600, bConfirm:= Confirmar);
	IntervCalibracao[3](evtEntry:= TC_Events.IntervaloExcedidoCalibracao.Calibracao_L3, bEvt:= DT_TO_UDINT(Main.HoraAtual) - HMI.UltimoAlrCalibr[3] > IntervaloLavCalibr.IntervaloCalibracao * 3600, bConfirm:= Confirmar);
	IntervCalibracao[4](evtEntry:= TC_Events.IntervaloExcedidoCalibracao.Calibracao_L4, bEvt:= DT_TO_UDINT(Main.HoraAtual) - HMI.UltimoAlrCalibr[4] > IntervaloLavCalibr.IntervaloCalibracao * 3600, bConfirm:= Confirmar);
	IntervCalibracao[5](evtEntry:= TC_Events.IntervaloExcedidoCalibracao.Calibracao_L5, bEvt:= DT_TO_UDINT(Main.HoraAtual) - HMI.UltimoAlrCalibr[5] > IntervaloLavCalibr.IntervaloCalibracao * 3600, bConfirm:= Confirmar);
	IntervCalibracao[6](evtEntry:= TC_Events.IntervaloExcedidoCalibracao.Calibracao_L6, bEvt:= DT_TO_UDINT(Main.HoraAtual) - HMI.UltimoAlrCalibr[6] > IntervaloLavCalibr.IntervaloCalibracao * 3600, bConfirm:= Confirmar);
	IntervCalibracao[7](evtEntry:= TC_Events.IntervaloExcedidoCalibracao.Calibracao_L7, bEvt:= DT_TO_UDINT(Main.HoraAtual) - HMI.UltimoAlrCalibr[7] > IntervaloLavCalibr.IntervaloCalibracao * 3600, bConfirm:= Confirmar);
	IntervCalibracao[8](evtEntry:= TC_Events.IntervaloExcedidoCalibracao.Calibracao_L8, bEvt:= DT_TO_UDINT(Main.HoraAtual) - HMI.UltimoAlrCalibr[8] > IntervaloLavCalibr.IntervaloCalibracao * 3600, bConfirm:= Confirmar);
	IntervCalibracao[9](evtEntry:= TC_Events.IntervaloExcedidoCalibracao.Calibracao_L9, bEvt:= DT_TO_UDINT(Main.HoraAtual) - HMI.UltimoAlrCalibr[9] > IntervaloLavCalibr.IntervaloCalibracao * 3600, bConfirm:= Confirmar);
	IntervCalibracao[10](evtEntry:= TC_Events.IntervaloExcedidoCalibracao.Calibracao_L10, bEvt:= DT_TO_UDINT(Main.HoraAtual) - HMI.UltimoAlrCalibr[10] > IntervaloLavCalibr.IntervaloCalibracao * 3600, bConfirm:= Confirmar);
	IntervCalibracao[11](evtEntry:= TC_Events.IntervaloExcedidoCalibracao.Calibracao_L11, bEvt:= DT_TO_UDINT(Main.HoraAtual) - HMI.UltimoAlrCalibr[11] > IntervaloLavCalibr.IntervaloCalibracao * 3600, bConfirm:= Confirmar);
	IntervCalibracao[12](evtEntry:= TC_Events.IntervaloExcedidoCalibracao.Calibracao_L12, bEvt:= DT_TO_UDINT(Main.HoraAtual) - HMI.UltimoAlrCalibr[12] > IntervaloLavCalibr.IntervaloCalibracao * 3600, bConfirm:= Confirmar);
{endregion}

{Region "Intervalo de lavagem excedido"}
	IntervLavagem[1](evtEntry:= TC_Events.IntervaloExcedidoLavagem.IntervaloExcedidoL1, bEvt:= (DT_TO_LINT(Main.HoraAtual) - Liquidos.UltimoAlrLavagem[1]) > IntervaloLavCalibr.IntervaloLavagem * 3600, bConfirm:= Confirmar);
	IntervLavagem[2](evtEntry:= TC_Events.IntervaloExcedidoLavagem.IntervaloExcedidoL2, bEvt:= (DT_TO_LINT(Main.HoraAtual) - Liquidos.UltimoAlrLavagem[2]) > IntervaloLavCalibr.IntervaloLavagem * 3600, bConfirm:= Confirmar);
	IntervLavagem[3](evtEntry:= TC_Events.IntervaloExcedidoLavagem.IntervaloExcedidoL3, bEvt:= (DT_TO_LINT(Main.HoraAtual) - Liquidos.UltimoAlrLavagem[3]) > IntervaloLavCalibr.IntervaloLavagem * 3600, bConfirm:= Confirmar);
	IntervLavagem[4](evtEntry:= TC_Events.IntervaloExcedidoLavagem.IntervaloExcedidoL4, bEvt:= (DT_TO_LINT(Main.HoraAtual) - Liquidos.UltimoAlrLavagem[4]) > IntervaloLavCalibr.IntervaloLavagem * 3600, bConfirm:= Confirmar);
	IntervLavagem[5](evtEntry:= TC_Events.IntervaloExcedidoLavagem.IntervaloExcedidoL5, bEvt:= (DT_TO_LINT(Main.HoraAtual) - Liquidos.UltimoAlrLavagem[5]) > IntervaloLavCalibr.IntervaloLavagem * 3600, bConfirm:= Confirmar);
	IntervLavagem[6](evtEntry:= TC_Events.IntervaloExcedidoLavagem.IntervaloExcedidoL6, bEvt:= (DT_TO_LINT(Main.HoraAtual) - Liquidos.UltimoAlrLavagem[6]) > IntervaloLavCalibr.IntervaloLavagem * 3600, bConfirm:= Confirmar);
	IntervLavagem[7](evtEntry:= TC_Events.IntervaloExcedidoLavagem.IntervaloExcedidoL7, bEvt:= (DT_TO_LINT(Main.HoraAtual) - Liquidos.UltimoAlrLavagem[7]) > IntervaloLavCalibr.IntervaloLavagem * 3600, bConfirm:= Confirmar);
	IntervLavagem[8](evtEntry:= TC_Events.IntervaloExcedidoLavagem.IntervaloExcedidoL8, bEvt:= (DT_TO_LINT(Main.HoraAtual) - Liquidos.UltimoAlrLavagem[8]) > IntervaloLavCalibr.IntervaloLavagem * 3600, bConfirm:= Confirmar);
	IntervLavagem[9](evtEntry:= TC_Events.IntervaloExcedidoLavagem.IntervaloExcedidoL9, bEvt:= (DT_TO_LINT(Main.HoraAtual) - Liquidos.UltimoAlrLavagem[9]) > IntervaloLavCalibr.IntervaloLavagem * 3600, bConfirm:= Confirmar);
	IntervLavagem[10](evtEntry:= TC_Events.IntervaloExcedidoLavagem.IntervaloExcedidoL10, bEvt:= (DT_TO_LINT(Main.HoraAtual) - Liquidos.UltimoAlrLavagem[10]) > IntervaloLavCalibr.IntervaloLavagem * 3600, bConfirm:= Confirmar);
	IntervLavagem[11](evtEntry:= TC_Events.IntervaloExcedidoLavagem.IntervaloExcedidoL11, bEvt:= (DT_TO_LINT(Main.HoraAtual) - Liquidos.UltimoAlrLavagem[11]) > IntervaloLavCalibr.IntervaloLavagem * 3600, bConfirm:= Confirmar);
	IntervLavagem[12](evtEntry:= TC_Events.IntervaloExcedidoLavagem.IntervaloExcedidoL12, bEvt:= (DT_TO_LINT(Main.HoraAtual) - Liquidos.UltimoAlrLavagem[12]) > IntervaloLavCalibr.IntervaloLavagem * 3600, bConfirm:= Confirmar);

{endregion}

{Region "Ângulo de abertura das válvulas IOLink"}
	//Válvula 1
	AnguloValv[1](evtEntry:= TC_Events.AnguloValvulas.AnguloV1L1, bEvt:= Circuito_L1.ControlValv_ioLink_V1.Range < RangeMinimo, bConfirm:= Confirmar);
	AnguloValv[2](evtEntry:= TC_Events.AnguloValvulas.AnguloV1L2, bEvt:= Circuito_L2.ControlValv_ioLink_V1.Range < RangeMinimo, bConfirm:= Confirmar);
	AnguloValv[3](evtEntry:= TC_Events.AnguloValvulas.AnguloV1L3, bEvt:= Circuito_L3.ControlValv_ioLink_V1.Range < RangeMinimo, bConfirm:= Confirmar);
	AnguloValv[4](evtEntry:= TC_Events.AnguloValvulas.AnguloV1L4, bEvt:= Circuito_L4.ControlValv_ioLink_V1.Range < RangeMinimo, bConfirm:= Confirmar);
	AnguloValv[5](evtEntry:= TC_Events.AnguloValvulas.AnguloV1L5, bEvt:= Circuito_L5.ControlValv_ioLink_V1.Range < RangeMinimo, bConfirm:= Confirmar);
	AnguloValv[6](evtEntry:= TC_Events.AnguloValvulas.AnguloV1L6, bEvt:= Circuito_L6.ControlValv_ioLink_V1.Range < RangeMinimo, bConfirm:= Confirmar);
	AnguloValv[7](evtEntry:= TC_Events.AnguloValvulas.AnguloV1L7, bEvt:= Circuito_L7.ControlValv_ioLink_V1.Range < RangeMinimo, bConfirm:= Confirmar);
	AnguloValv[8](evtEntry:= TC_Events.AnguloValvulas.AnguloV1L8, bEvt:= Circuito_L8.ControlValv_ioLink_V1.Range < RangeMinimo, bConfirm:= Confirmar);
	AnguloValv[9](evtEntry:= TC_Events.AnguloValvulas.AnguloV1L9, bEvt:= Circuito_L9.ControlValv_ioLink_V1.Range < RangeMinimo, bConfirm:= Confirmar);
	AnguloValv[10](evtEntry:= TC_Events.AnguloValvulas.AnguloV1L10, bEvt:= Circuito_L10.ControlValv_ioLink_V1.Range < RangeMinimo, bConfirm:= Confirmar);
	AnguloValv[11](evtEntry:= TC_Events.AnguloValvulas.AnguloV1L11, bEvt:= Circuito_L11.ControlValv_ioLink_V1.Range < RangeMinimo, bConfirm:= Confirmar);
	AnguloValv[12](evtEntry:= TC_Events.AnguloValvulas.AnguloV1L12, bEvt:= Circuito_L12.ControlValv_ioLink_V1.Range < RangeMinimo, bConfirm:= Confirmar);
	
	//Válvula 2
	AnguloValv[13](evtEntry:= TC_Events.AnguloValvulas.AnguloV2L1, bEvt:= Circuito_L1.ControlValv_ioLink_V2.Range < RangeMinimo, bConfirm:= Confirmar);
	AnguloValv[14](evtEntry:= TC_Events.AnguloValvulas.AnguloV2L2, bEvt:= Circuito_L2.ControlValv_ioLink_V2.Range < RangeMinimo, bConfirm:= Confirmar);
	AnguloValv[15](evtEntry:= TC_Events.AnguloValvulas.AnguloV2L3, bEvt:= Circuito_L3.ControlValv_ioLink_V2.Range < RangeMinimo, bConfirm:= Confirmar);
	AnguloValv[16](evtEntry:= TC_Events.AnguloValvulas.AnguloV2L4, bEvt:= Circuito_L4.ControlValv_ioLink_V2.Range < RangeMinimo, bConfirm:= Confirmar);
	AnguloValv[17](evtEntry:= TC_Events.AnguloValvulas.AnguloV2L5, bEvt:= Circuito_L5.ControlValv_ioLink_V2.Range < RangeMinimo, bConfirm:= Confirmar);
	AnguloValv[18](evtEntry:= TC_Events.AnguloValvulas.AnguloV2L6, bEvt:= Circuito_L6.ControlValv_ioLink_V2.Range < RangeMinimo, bConfirm:= Confirmar);
	AnguloValv[19](evtEntry:= TC_Events.AnguloValvulas.AnguloV2L7, bEvt:= Circuito_L7.ControlValv_ioLink_V2.Range < RangeMinimo, bConfirm:= Confirmar);
	AnguloValv[20](evtEntry:= TC_Events.AnguloValvulas.AnguloV2L8, bEvt:= Circuito_L8.ControlValv_ioLink_V2.Range < RangeMinimo, bConfirm:= Confirmar);
	AnguloValv[21](evtEntry:= TC_Events.AnguloValvulas.AnguloV2L9, bEvt:= Circuito_L9.ControlValv_ioLink_V2.Range < RangeMinimo, bConfirm:= Confirmar);
	AnguloValv[22](evtEntry:= TC_Events.AnguloValvulas.AnguloV2L10, bEvt:= Circuito_L10.ControlValv_ioLink_V2.Range < RangeMinimo, bConfirm:= Confirmar);
	AnguloValv[23](evtEntry:= TC_Events.AnguloValvulas.AnguloV2L11, bEvt:= Circuito_L11.ControlValv_ioLink_V2.Range < RangeMinimo, bConfirm:= Confirmar);
	AnguloValv[24](evtEntry:= TC_Events.AnguloValvulas.AnguloV2L12, bEvt:= Circuito_L12.ControlValv_ioLink_V2.Range < RangeMinimo, bConfirm:= Confirmar);
	
	//Válvula 3
	AnguloValv[25](evtEntry:= TC_Events.AnguloValvulas.AnguloV3L1, bEvt:= Circuito_L1.ControlValv_ioLink_V3.Range < RangeMinimo, bConfirm:= Confirmar);
	AnguloValv[26](evtEntry:= TC_Events.AnguloValvulas.AnguloV3L2, bEvt:= Circuito_L2.ControlValv_ioLink_V3.Range < RangeMinimo, bConfirm:= Confirmar);
	AnguloValv[27](evtEntry:= TC_Events.AnguloValvulas.AnguloV3L3, bEvt:= Circuito_L3.ControlValv_ioLink_V3.Range < RangeMinimo, bConfirm:= Confirmar);
	AnguloValv[28](evtEntry:= TC_Events.AnguloValvulas.AnguloV3L4, bEvt:= Circuito_L4.ControlValv_ioLink_V3.Range < RangeMinimo, bConfirm:= Confirmar);
	AnguloValv[29](evtEntry:= TC_Events.AnguloValvulas.AnguloV3L5, bEvt:= Circuito_L5.ControlValv_ioLink_V3.Range < RangeMinimo, bConfirm:= Confirmar);
	AnguloValv[30](evtEntry:= TC_Events.AnguloValvulas.AnguloV3L6, bEvt:= Circuito_L6.ControlValv_ioLink_V3.Range < RangeMinimo, bConfirm:= Confirmar);
	AnguloValv[31](evtEntry:= TC_Events.AnguloValvulas.AnguloV3L7, bEvt:= Circuito_L7.ControlValv_ioLink_V3.Range < RangeMinimo, bConfirm:= Confirmar);
	AnguloValv[32](evtEntry:= TC_Events.AnguloValvulas.AnguloV3L8, bEvt:= Circuito_L8.ControlValv_ioLink_V3.Range < RangeMinimo, bConfirm:= Confirmar);
	AnguloValv[33](evtEntry:= TC_Events.AnguloValvulas.AnguloV3L9, bEvt:= Circuito_L9.ControlValv_ioLink_V3.Range < RangeMinimo, bConfirm:= Confirmar);
	AnguloValv[34](evtEntry:= TC_Events.AnguloValvulas.AnguloV3L10, bEvt:= Circuito_L10.ControlValv_ioLink_V3.Range < RangeMinimo, bConfirm:= Confirmar);
	AnguloValv[35](evtEntry:= TC_Events.AnguloValvulas.AnguloV3L11, bEvt:= Circuito_L11.ControlValv_ioLink_V3.Range < RangeMinimo, bConfirm:= Confirmar);
	AnguloValv[36](evtEntry:= TC_Events.AnguloValvulas.AnguloV3L12, bEvt:= Circuito_L12.ControlValv_ioLink_V3.Range < RangeMinimo, bConfirm:= Confirmar);
	
	//Válvula 4
	AnguloValv[37](evtEntry:= TC_Events.AnguloValvulas.AnguloV4L1, bEvt:= Circuito_L1.ControlValv_ioLink_V4.Range < RangeMinimo, bConfirm:= Confirmar);
	AnguloValv[38](evtEntry:= TC_Events.AnguloValvulas.AnguloV4L2, bEvt:= Circuito_L2.ControlValv_ioLink_V4.Range < RangeMinimo, bConfirm:= Confirmar);
	AnguloValv[39](evtEntry:= TC_Events.AnguloValvulas.AnguloV4L3, bEvt:= Circuito_L3.ControlValv_ioLink_V4.Range < RangeMinimo, bConfirm:= Confirmar);
	AnguloValv[40](evtEntry:= TC_Events.AnguloValvulas.AnguloV4L4, bEvt:= Circuito_L4.ControlValv_ioLink_V4.Range < RangeMinimo, bConfirm:= Confirmar);
	AnguloValv[41](evtEntry:= TC_Events.AnguloValvulas.AnguloV4L5, bEvt:= Circuito_L5.ControlValv_ioLink_V4.Range < RangeMinimo, bConfirm:= Confirmar);
	AnguloValv[42](evtEntry:= TC_Events.AnguloValvulas.AnguloV4L6, bEvt:= Circuito_L6.ControlValv_ioLink_V4.Range < RangeMinimo, bConfirm:= Confirmar);
	AnguloValv[43](evtEntry:= TC_Events.AnguloValvulas.AnguloV4L7, bEvt:= Circuito_L7.ControlValv_ioLink_V4.Range < RangeMinimo, bConfirm:= Confirmar);
	AnguloValv[44](evtEntry:= TC_Events.AnguloValvulas.AnguloV4L8, bEvt:= Circuito_L8.ControlValv_ioLink_V4.Range < RangeMinimo, bConfirm:= Confirmar);
	AnguloValv[45](evtEntry:= TC_Events.AnguloValvulas.AnguloV4L9, bEvt:= Circuito_L9.ControlValv_ioLink_V4.Range < RangeMinimo, bConfirm:= Confirmar);
	AnguloValv[46](evtEntry:= TC_Events.AnguloValvulas.AnguloV4L10, bEvt:= Circuito_L10.ControlValv_ioLink_V4.Range < RangeMinimo, bConfirm:= Confirmar);
	AnguloValv[47](evtEntry:= TC_Events.AnguloValvulas.AnguloV4L11, bEvt:= Circuito_L11.ControlValv_ioLink_V4.Range < RangeMinimo, bConfirm:= Confirmar);
	AnguloValv[48](evtEntry:= TC_Events.AnguloValvulas.AnguloV4L12, bEvt:= Circuito_L12.ControlValv_ioLink_V4.Range < RangeMinimo, bConfirm:= Confirmar);
{endregion}

{Region "Diagnósticos do iPC"}
	iPC_Diag[1](evtEntry:= TC_Events.iPC_Diagnostic.UsoCPU, bEvt:= Ipc_Diagnostic.CpuUsage > 90, bConfirm:= Confirmar);
	iPC_Diag[2](evtEntry:= TC_Events.iPC_Diagnostic.DiscoRigido, bEvt:= (Ipc_Diagnostic.rDiskTotalSize-iPC_Diagnostic.rFreeDisk)/(Ipc_Diagnostic.rDiskTotalSize+0.01) > 90, bConfirm:= Confirmar);
	iPC_Diag[3](evtEntry:= TC_Events.iPC_Diagnostic.MemoriaRAM, bEvt:= (Ipc_Diagnostic.rTotalRAM-iPC_Diagnostic.rFreeRAM)/(Ipc_Diagnostic.rTotalRAM+0.01) > 90, bConfirm:= Confirmar);
	iPC_Diag[4](evtEntry:= TC_Events.iPC_Diagnostic.TemperaturaCPU, bEvt:= Ipc_Diagnostic.CpuTemp > (0.9*TO_REAL(iPC_Diagnostic.MB_MaxTemperature)), bConfirm:= Confirmar);
	iPC_Diag[5](evtEntry:= TC_Events.iPC_Diagnostic.TemperaturaPlacaMae, bEvt:= Ipc_Diagnostic.MB_Temperature > (0.9*TO_REAL(iPC_Diagnostic.MB_MaxTemperature)), bConfirm:= Confirmar);
{endregion}

{Region "Nível baixo dos produtos"}
	NivelProd[1](evtEntry:= TC_Events.BaixoNivelPoLiq.BaixoNivelLIQ1, bEvt:= Entradas.PU1_WT1_rValue_REAL < 50, bConfirm:= Confirmar);
	NivelProd[2](evtEntry:= TC_Events.BaixoNivelPoLiq.BaixoNivelLIQ2, bEvt:= Entradas.PU1_WT2_rValue_REAL < 50, bConfirm:= Confirmar);
	NivelProd[3](evtEntry:= TC_Events.BaixoNivelPoLiq.BaixoNivelLIQ3, bEvt:= Entradas.PU1_WT3_rValue_REAL < 50, bConfirm:= Confirmar);
	NivelProd[4](evtEntry:= TC_Events.BaixoNivelPoLiq.BaixoNivelLIQ4, bEvt:= Entradas.PU1_WT4_rValue_REAL < 50, bConfirm:= Confirmar);
	NivelProd[5](evtEntry:= TC_Events.BaixoNivelPoLiq.BaixoNivelLIQ5, bEvt:= Entradas.PU2_WT5_rValue_REAL < 50, bConfirm:= Confirmar);
	NivelProd[6](evtEntry:= TC_Events.BaixoNivelPoLiq.BaixoNivelLIQ6, bEvt:= Entradas.PU2_WT6_rValue_REAL < 50, bConfirm:= Confirmar);
	NivelProd[7](evtEntry:= TC_Events.BaixoNivelPoLiq.BaixoNivelLIQ7, bEvt:= Entradas.PU2_WT7_rValue_REAL < 50, bConfirm:= Confirmar);
	NivelProd[8](evtEntry:= TC_Events.BaixoNivelPoLiq.BaixoNivelLIQ8, bEvt:= Entradas.PU2_WT8_rValue_REAL < 50, bConfirm:= Confirmar);
	NivelProd[9](evtEntry:= TC_Events.BaixoNivelPoLiq.BaixoNivelLIQ9, bEvt:= Entradas.PU3_WT9_rValue_REAL < 50, bConfirm:= Confirmar);
	NivelProd[10](evtEntry:= TC_Events.BaixoNivelPoLiq.BaixoNivelLIQ10, bEvt:= Entradas.PU3_WT10_rValue_REAL < 50, bConfirm:= Confirmar);
	NivelProd[11](evtEntry:= TC_Events.BaixoNivelPoLiq.BaixoNivelLIQ11, bEvt:= Entradas.PU3_WT11_rValue_REAL < 50, bConfirm:= Confirmar);
	NivelProd[12](evtEntry:= TC_Events.BaixoNivelPoLiq.BaixoNivelLIQ12, bEvt:= Entradas.PU3_WT12_rValue_REAL < 50, bConfirm:= Confirmar);
	NivelProd[13](evtEntry:= TC_Events.BaixoNivelPoLiq.BaixoNivelPO1, bEvt:= entradas.TR_P1_LLS, bConfirm:= Confirmar);
	NivelProd[14](evtEntry:= TC_Events.BaixoNivelPoLiq.BaixoNivelPO2, bEvt:= entradas.TR_P2_LLS, bConfirm:= Confirmar);
{endregion}

END_PROGRAM

// ---- POUs/Testes Thiago/GeraAlarme.TcPOU
FUNCTION_BLOCK GeraAlarme EXTENDS FB_TcAlarm
VAR_INPUT
	evtEntry:tcEventEntry;
	bEvt:BOOL;
	bConfirm:BOOL;
END_VAR
VAR_OUTPUT
END_VAR
VAR
	bInit:BOOL:=TRUE;
	bMem:BOOL;
END_VAR

IF bInit THEN
	SUPER^.CreateEx(evtEntry, TRUE, 0);
	bInit := FALSE;
END_IF

IF bEvt AND  NOT bMem AND SUPER^.eConfirmationState <> tcEventConfirmationState.WaitForConfirmation THEN
	SUPER^.Raise(0);
END_IF

IF bMem AND NOT bEvt THEN
	SUPER^.Clear(0,FALSE);
END_IF

IF bConfirm THEN
	SUPER^.Confirm(0);
END_IF
bMem := bEvt;

END_FUNCTION_BLOCK

// ---- POUs/Agitadores.TcPOU
PROGRAM Agitadores
VAR
	PP1_L1_AG: Equipo_Motor_No_Rev;
	wPP1_L1_AG_HoraIni:INT;
	wPP1_L1_AG_CantHora:INT;
	wPP1_L1_AG_HoraFin:INT;
	bPP1_L1_AG_ResetAl: BOOL;	
	//
	PP1_L2_AG: Equipo_Motor_No_Rev;
	wPP1_L2_AG_HoraIni:INT;
	wPP1_L2_AG_CantHora:INT;
	wPP1_L2_AG_HoraFin:INT;
	//
	PP1_L3_AG: Equipo_Motor_No_Rev;
	wPP1_L3_AG_HoraIni:INT;
	wPP1_L3_AG_CantHora:INT;
	wPP1_L3_AG_HoraFin:INT;	
	//
	PP1_L4_AG: Equipo_Motor_No_Rev;
	wPP1_L4_AG_HoraIni:INT;
	wPP1_L4_AG_CantHora:INT;
	wPP1_L4_AG_HoraFin:INT;	
	//	
	PP2_L5_AG: Equipo_Motor_No_Rev;
	wPP2_L5_AG_HoraIni:INT;
	wPP2_L5_AG_CantHora:INT;
	wPP2_L5_AG_HoraFin:INT;
	bPP2_L5_AG_ResetAl: BOOL;	
	//
	PP2_L6_AG: Equipo_Motor_No_Rev;
	wPP2_L6_AG_HoraIni:INT;
	wPP2_L6_AG_CantHora:INT;
	wPP2_L6_AG_HoraFin:INT;	
	//
	PP2_L7_AG: Equipo_Motor_No_Rev;
	wPP2_L7_AG_HoraIni:INT;
	wPP2_L7_AG_CantHora:INT;
	wPP2_L7_AG_HoraFin:INT;	
	//
	PP2_L8_AG: Equipo_Motor_No_Rev;
	wPP2_L8_AG_HoraIni:INT;
	wPP2_L8_AG_CantHora:INT;
	wPP2_L8_AG_HoraFin:INT;
	//
	PP3_L9_AG: Equipo_Motor_No_Rev;
	wPP3_L9_AG_HoraIni:INT;
	wPP3_L9_AG_CantHora:INT;
	wPP3_L9_AG_HoraFin:INT;	
	//
	PP3_L10_AG: Equipo_Motor_No_Rev;
	wPP3_L10_AG_HoraIni:INT;
	wPP3_L10_AG_CantHora:INT;
	wPP3_L10_AG_HoraFin:INT;	
	//
	PP3_L11_AG: Equipo_Motor_No_Rev;
	wPP3_L11_AG_HoraIni:INT;
	wPP3_L11_AG_CantHora:INT;
	wPP3_L11_AG_HoraFin:INT;	
	//
	PP3_L12_AG: Equipo_Motor_No_Rev;
	wPP3_L12_AG_HoraIni:INT;
	wPP3_L12_AG_CantHora:INT;
	wPP3_L12_AG_HoraFin:INT;	
END_VAR

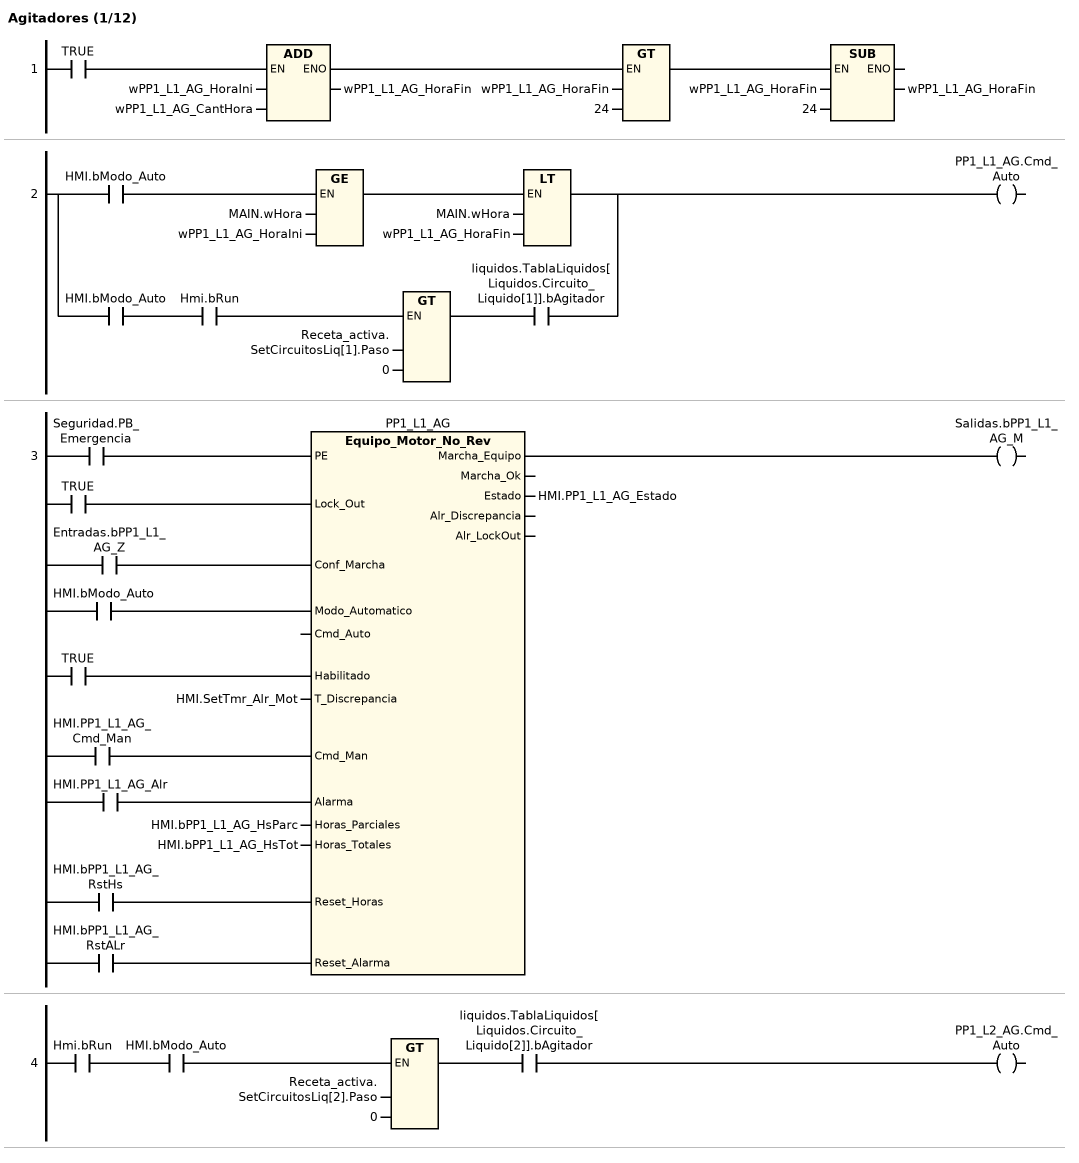
// NETWORK 1
wPP1_L1_AG_HoraFin := wPP1_L1_AG_HoraIni + wPP1_L1_AG_CantHora;
IF wPP1_L1_AG_HoraFin > 24 THEN wPP1_L1_AG_HoraFin := wPP1_L1_AG_HoraFin - 24; END_IF

// NETWORK 2
PP1_L1_AG.Cmd_Auto := HMI.bModo_Auto AND MAIN.wHora >= wPP1_L1_AG_HoraIni AND MAIN.wHora < wPP1_L1_AG_HoraFin OR (HMI.bModo_Auto AND Hmi.bRun AND Receta_activa.SetCircuitosLiq[1].Paso > 0) AND (liquidos.TablaLiquidos[Liquidos.Circuito_Liquido[1]].bAgitador);

// NETWORK 3
PP1_L1_AG(
    PE := Seguridad.PB_Emergencia,
    Lock_Out := TRUE,
    Conf_Marcha := Entradas.bPP1_L1_AG_Z,
    Modo_Automatico := HMI.bModo_Auto,
    Habilitado := TRUE,
    T_Discrepancia := HMI.SetTmr_Alr_Mot,
    Cmd_Man := HMI.PP1_L1_AG_Cmd_Man,
    Alarma := HMI.PP1_L1_AG_Alr,
    Horas_Parciales := HMI.bPP1_L1_AG_HsParc,
    Horas_Totales := HMI.bPP1_L1_AG_HsTot,
    Reset_Horas := HMI.bPP1_L1_AG_RstHs,
    Reset_Alarma := HMI.bPP1_L1_AG_RstALr,
    Estado => HMI.PP1_L1_AG_Estado); // Equipo_Motor_No_Rev
Salidas.bPP1_L1_AG_M := PP1_L1_AG.Marcha_Equipo;

// NETWORK 4
PP1_L2_AG.Cmd_Auto := (Hmi.bRun AND HMI.bModo_Auto AND Receta_activa.SetCircuitosLiq[2].Paso > 0) AND (liquidos.TablaLiquidos[Liquidos.Circuito_Liquido[2]].bAgitador);

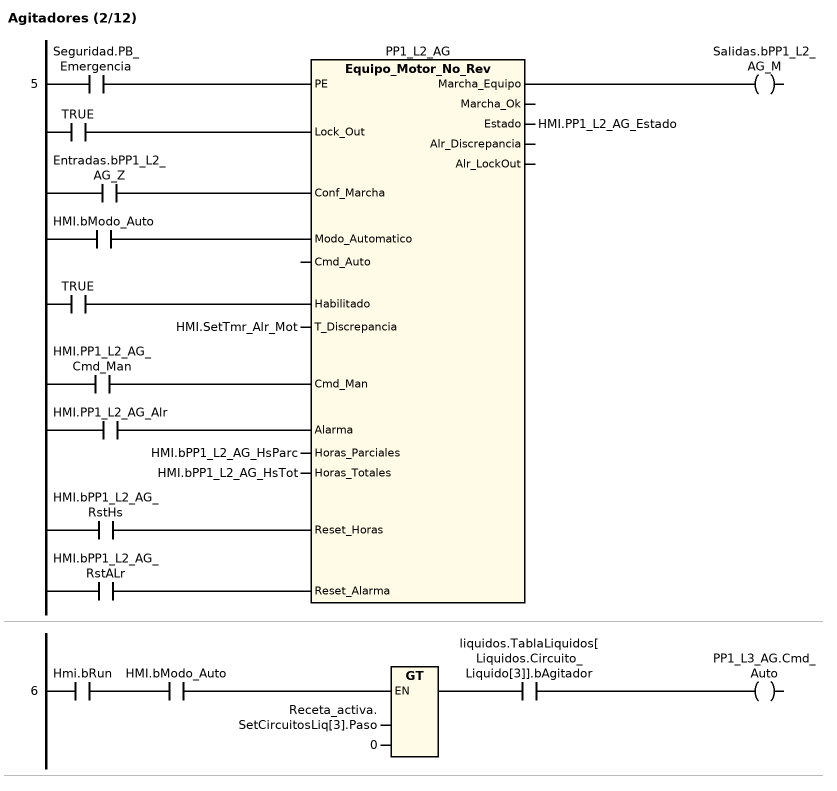
// NETWORK 5
PP1_L2_AG(
    PE := Seguridad.PB_Emergencia,
    Lock_Out := TRUE,
    Conf_Marcha := Entradas.bPP1_L2_AG_Z,
    Modo_Automatico := HMI.bModo_Auto,
    Habilitado := TRUE,
    T_Discrepancia := HMI.SetTmr_Alr_Mot,
    Cmd_Man := HMI.PP1_L2_AG_Cmd_Man,
    Alarma := HMI.PP1_L2_AG_Alr,
    Horas_Parciales := HMI.bPP1_L2_AG_HsParc,
    Horas_Totales := HMI.bPP1_L2_AG_HsTot,
    Reset_Horas := HMI.bPP1_L2_AG_RstHs,
    Reset_Alarma := HMI.bPP1_L2_AG_RstALr,
    Estado => HMI.PP1_L2_AG_Estado); // Equipo_Motor_No_Rev
Salidas.bPP1_L2_AG_M := PP1_L2_AG.Marcha_Equipo;

// NETWORK 6
PP1_L3_AG.Cmd_Auto := (Hmi.bRun AND HMI.bModo_Auto AND Receta_activa.SetCircuitosLiq[3].Paso > 0) AND (liquidos.TablaLiquidos[Liquidos.Circuito_Liquido[3]].bAgitador);

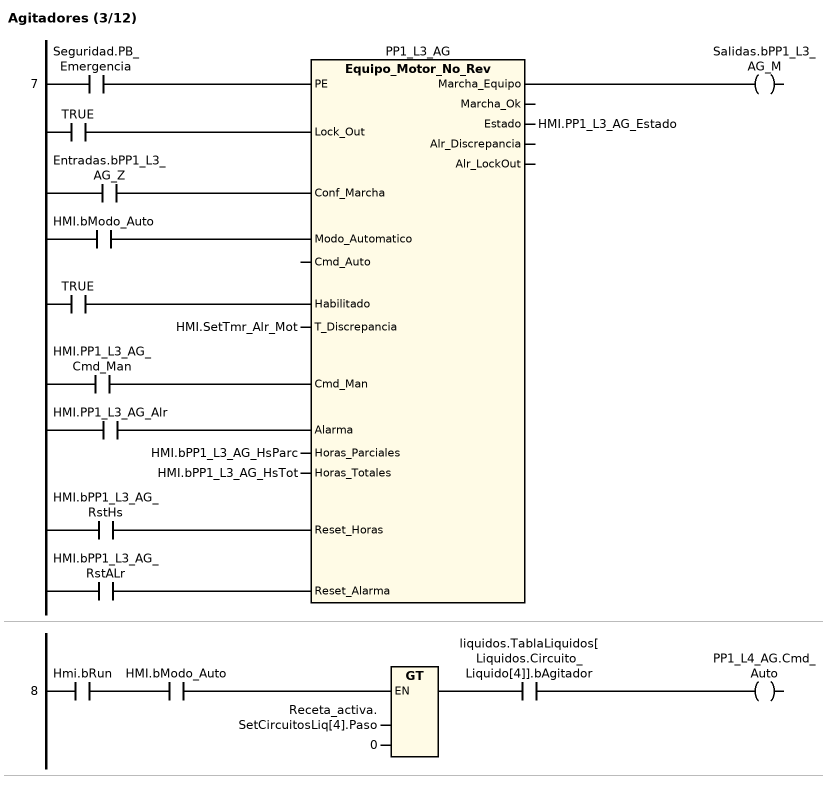
// NETWORK 7
PP1_L3_AG(
    PE := Seguridad.PB_Emergencia,
    Lock_Out := TRUE,
    Conf_Marcha := Entradas.bPP1_L3_AG_Z,
    Modo_Automatico := HMI.bModo_Auto,
    Habilitado := TRUE,
    T_Discrepancia := HMI.SetTmr_Alr_Mot,
    Cmd_Man := HMI.PP1_L3_AG_Cmd_Man,
    Alarma := HMI.PP1_L3_AG_Alr,
    Horas_Parciales := HMI.bPP1_L3_AG_HsParc,
    Horas_Totales := HMI.bPP1_L3_AG_HsTot,
    Reset_Horas := HMI.bPP1_L3_AG_RstHs,
    Reset_Alarma := HMI.bPP1_L3_AG_RstALr,
    Estado => HMI.PP1_L3_AG_Estado); // Equipo_Motor_No_Rev
Salidas.bPP1_L3_AG_M := PP1_L3_AG.Marcha_Equipo;

// NETWORK 8
PP1_L4_AG.Cmd_Auto := (Hmi.bRun AND HMI.bModo_Auto AND Receta_activa.SetCircuitosLiq[4].Paso > 0) AND (liquidos.TablaLiquidos[Liquidos.Circuito_Liquido[4]].bAgitador);

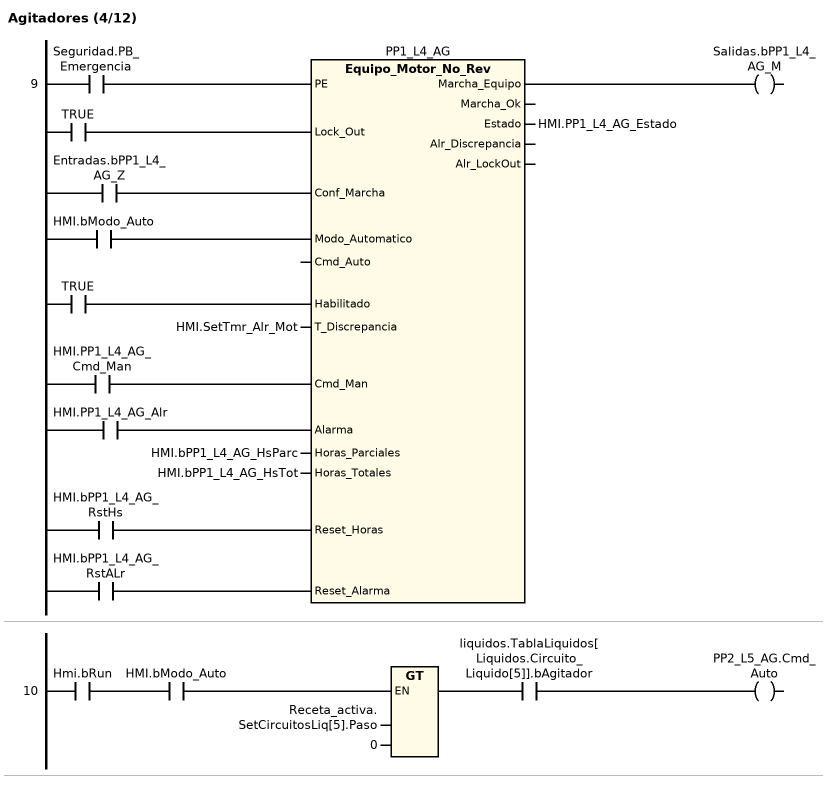
// NETWORK 9
PP1_L4_AG(
    PE := Seguridad.PB_Emergencia,
    Lock_Out := TRUE,
    Conf_Marcha := Entradas.bPP1_L4_AG_Z,
    Modo_Automatico := HMI.bModo_Auto,
    Habilitado := TRUE,
    T_Discrepancia := HMI.SetTmr_Alr_Mot,
    Cmd_Man := HMI.PP1_L4_AG_Cmd_Man,
    Alarma := HMI.PP1_L4_AG_Alr,
    Horas_Parciales := HMI.bPP1_L4_AG_HsParc,
    Horas_Totales := HMI.bPP1_L4_AG_HsTot,
    Reset_Horas := HMI.bPP1_L4_AG_RstHs,
    Reset_Alarma := HMI.bPP1_L4_AG_RstALr,
    Estado => HMI.PP1_L4_AG_Estado); // Equipo_Motor_No_Rev
Salidas.bPP1_L4_AG_M := PP1_L4_AG.Marcha_Equipo;

// NETWORK 10
PP2_L5_AG.Cmd_Auto := (Hmi.bRun AND HMI.bModo_Auto AND Receta_activa.SetCircuitosLiq[5].Paso > 0) AND (liquidos.TablaLiquidos[Liquidos.Circuito_Liquido[5]].bAgitador);

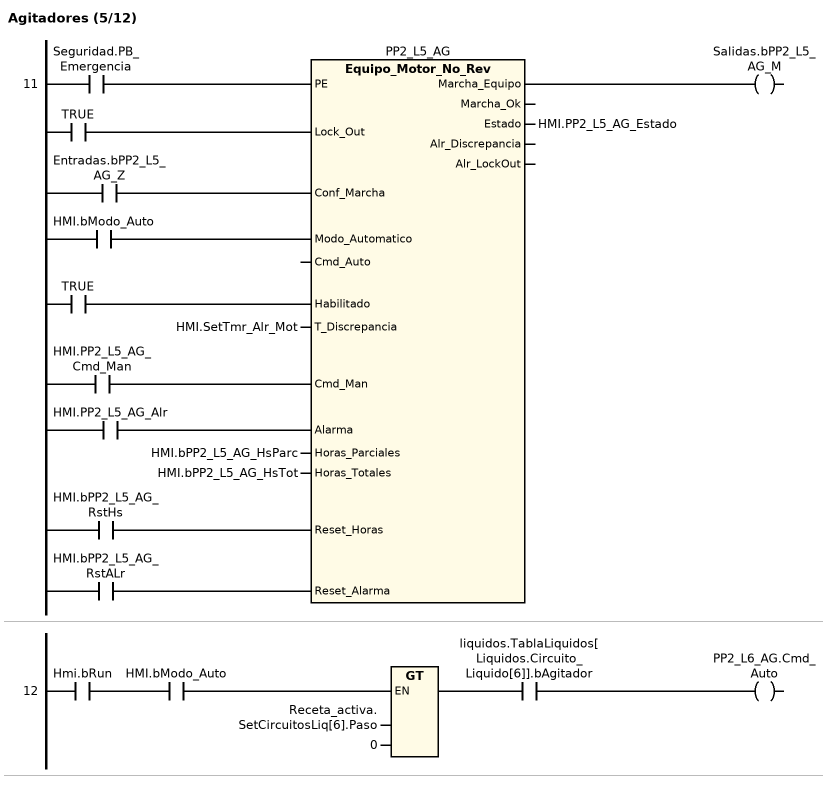
// NETWORK 11
PP2_L5_AG(
    PE := Seguridad.PB_Emergencia,
    Lock_Out := TRUE,
    Conf_Marcha := Entradas.bPP2_L5_AG_Z,
    Modo_Automatico := HMI.bModo_Auto,
    Habilitado := TRUE,
    T_Discrepancia := HMI.SetTmr_Alr_Mot,
    Cmd_Man := HMI.PP2_L5_AG_Cmd_Man,
    Alarma := HMI.PP2_L5_AG_Alr,
    Horas_Parciales := HMI.bPP2_L5_AG_HsParc,
    Horas_Totales := HMI.bPP2_L5_AG_HsTot,
    Reset_Horas := HMI.bPP2_L5_AG_RstHs,
    Reset_Alarma := HMI.bPP2_L5_AG_RstALr,
    Estado => HMI.PP2_L5_AG_Estado); // Equipo_Motor_No_Rev
Salidas.bPP2_L5_AG_M := PP2_L5_AG.Marcha_Equipo;

// NETWORK 12
PP2_L6_AG.Cmd_Auto := (Hmi.bRun AND HMI.bModo_Auto AND Receta_activa.SetCircuitosLiq[6].Paso > 0) AND (liquidos.TablaLiquidos[Liquidos.Circuito_Liquido[6]].bAgitador);

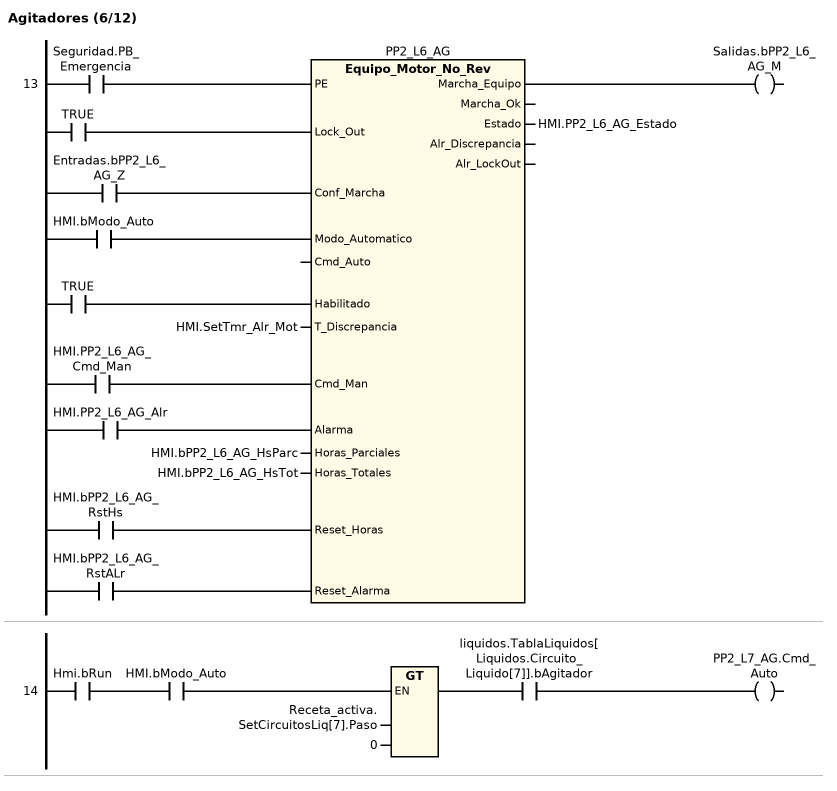
// NETWORK 13
PP2_L6_AG(
    PE := Seguridad.PB_Emergencia,
    Lock_Out := TRUE,
    Conf_Marcha := Entradas.bPP2_L6_AG_Z,
    Modo_Automatico := HMI.bModo_Auto,
    Habilitado := TRUE,
    T_Discrepancia := HMI.SetTmr_Alr_Mot,
    Cmd_Man := HMI.PP2_L6_AG_Cmd_Man,
    Alarma := HMI.PP2_L6_AG_Alr,
    Horas_Parciales := HMI.bPP2_L6_AG_HsParc,
    Horas_Totales := HMI.bPP2_L6_AG_HsTot,
    Reset_Horas := HMI.bPP2_L6_AG_RstHs,
    Reset_Alarma := HMI.bPP2_L6_AG_RstALr,
    Estado => HMI.PP2_L6_AG_Estado); // Equipo_Motor_No_Rev
Salidas.bPP2_L6_AG_M := PP2_L6_AG.Marcha_Equipo;

// NETWORK 14
PP2_L7_AG.Cmd_Auto := (Hmi.bRun AND HMI.bModo_Auto AND Receta_activa.SetCircuitosLiq[7].Paso > 0) AND (liquidos.TablaLiquidos[Liquidos.Circuito_Liquido[7]].bAgitador);

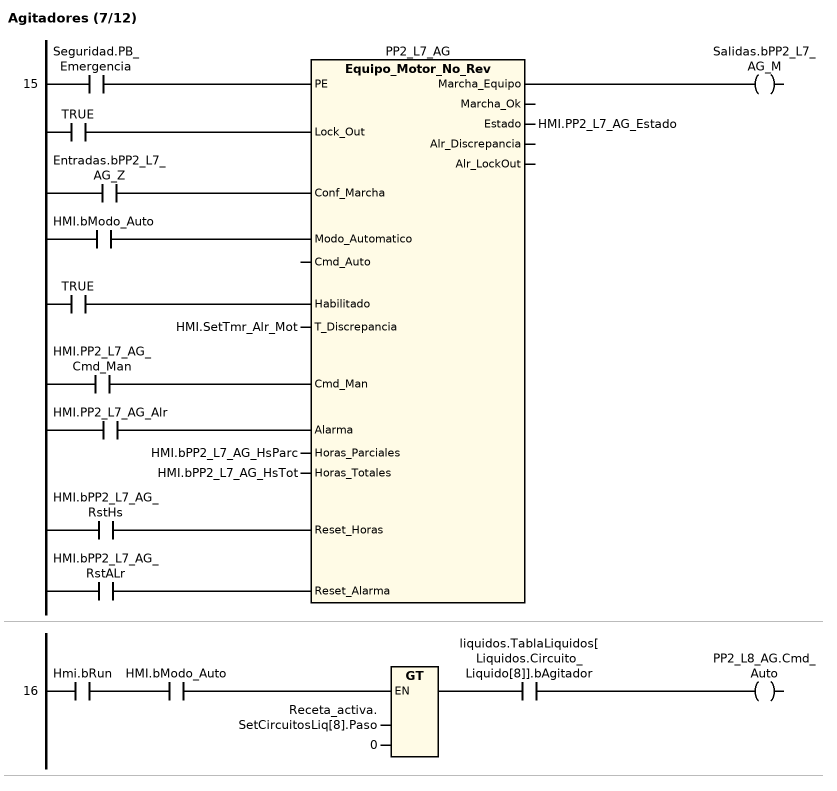
// NETWORK 15
PP2_L7_AG(
    PE := Seguridad.PB_Emergencia,
    Lock_Out := TRUE,
    Conf_Marcha := Entradas.bPP2_L7_AG_Z,
    Modo_Automatico := HMI.bModo_Auto,
    Habilitado := TRUE,
    T_Discrepancia := HMI.SetTmr_Alr_Mot,
    Cmd_Man := HMI.PP2_L7_AG_Cmd_Man,
    Alarma := HMI.PP2_L7_AG_Alr,
    Horas_Parciales := HMI.bPP2_L7_AG_HsParc,
    Horas_Totales := HMI.bPP2_L7_AG_HsTot,
    Reset_Horas := HMI.bPP2_L7_AG_RstHs,
    Reset_Alarma := HMI.bPP2_L7_AG_RstALr,
    Estado => HMI.PP2_L7_AG_Estado); // Equipo_Motor_No_Rev
Salidas.bPP2_L7_AG_M := PP2_L7_AG.Marcha_Equipo;

// NETWORK 16
PP2_L8_AG.Cmd_Auto := (Hmi.bRun AND HMI.bModo_Auto AND Receta_activa.SetCircuitosLiq[8].Paso > 0) AND (liquidos.TablaLiquidos[Liquidos.Circuito_Liquido[8]].bAgitador);

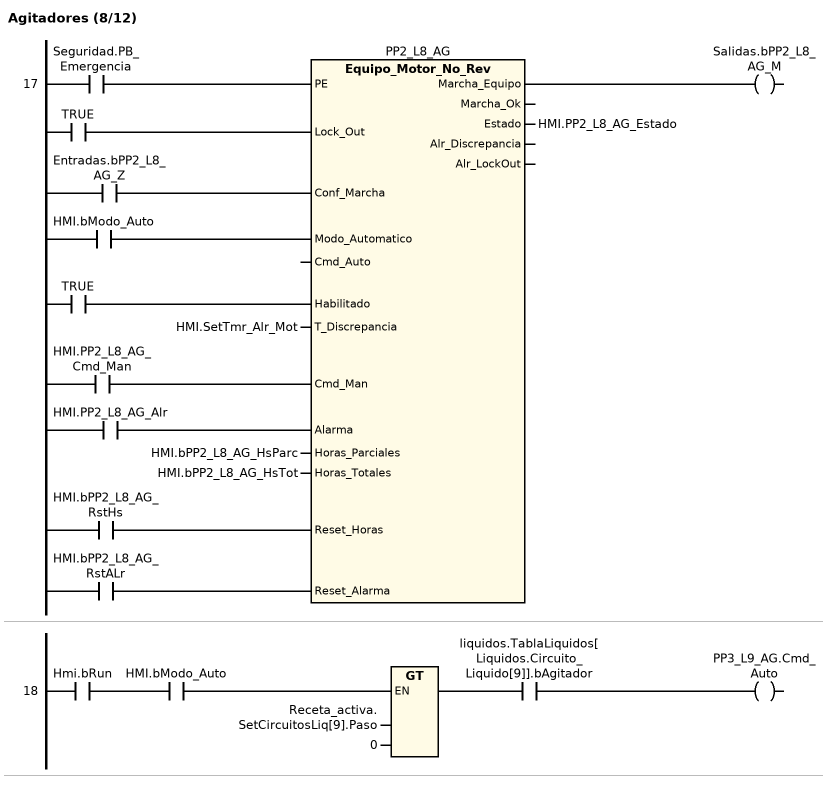
// NETWORK 17
PP2_L8_AG(
    PE := Seguridad.PB_Emergencia,
    Lock_Out := TRUE,
    Conf_Marcha := Entradas.bPP2_L8_AG_Z,
    Modo_Automatico := HMI.bModo_Auto,
    Habilitado := TRUE,
    T_Discrepancia := HMI.SetTmr_Alr_Mot,
    Cmd_Man := HMI.PP2_L8_AG_Cmd_Man,
    Alarma := HMI.PP2_L8_AG_Alr,
    Horas_Parciales := HMI.bPP2_L8_AG_HsParc,
    Horas_Totales := HMI.bPP2_L8_AG_HsTot,
    Reset_Horas := HMI.bPP2_L8_AG_RstHs,
    Reset_Alarma := HMI.bPP2_L8_AG_RstALr,
    Estado => HMI.PP2_L8_AG_Estado); // Equipo_Motor_No_Rev
Salidas.bPP2_L8_AG_M := PP2_L8_AG.Marcha_Equipo;

// NETWORK 18
PP3_L9_AG.Cmd_Auto := (Hmi.bRun AND HMI.bModo_Auto AND Receta_activa.SetCircuitosLiq[9].Paso > 0) AND (liquidos.TablaLiquidos[Liquidos.Circuito_Liquido[9]].bAgitador);

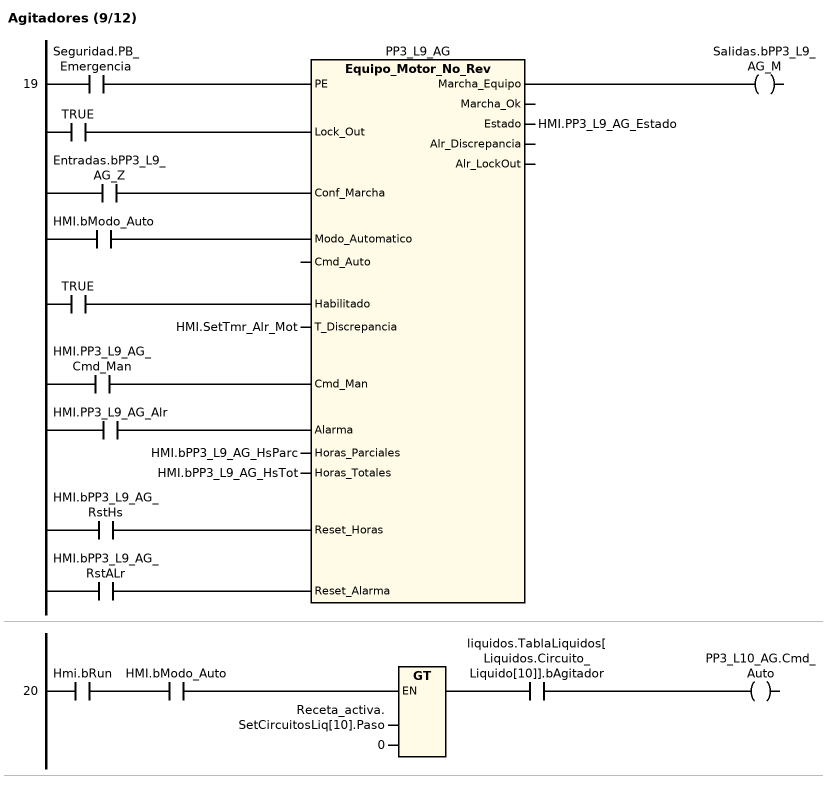
// NETWORK 19
PP3_L9_AG(
    PE := Seguridad.PB_Emergencia,
    Lock_Out := TRUE,
    Conf_Marcha := Entradas.bPP3_L9_AG_Z,
    Modo_Automatico := HMI.bModo_Auto,
    Habilitado := TRUE,
    T_Discrepancia := HMI.SetTmr_Alr_Mot,
    Cmd_Man := HMI.PP3_L9_AG_Cmd_Man,
    Alarma := HMI.PP3_L9_AG_Alr,
    Horas_Parciales := HMI.bPP3_L9_AG_HsParc,
    Horas_Totales := HMI.bPP3_L9_AG_HsTot,
    Reset_Horas := HMI.bPP3_L9_AG_RstHs,
    Reset_Alarma := HMI.bPP3_L9_AG_RstALr,
    Estado => HMI.PP3_L9_AG_Estado); // Equipo_Motor_No_Rev
Salidas.bPP3_L9_AG_M := PP3_L9_AG.Marcha_Equipo;

// NETWORK 20
PP3_L10_AG.Cmd_Auto := (Hmi.bRun AND HMI.bModo_Auto AND Receta_activa.SetCircuitosLiq[10].Paso > 0) AND (liquidos.TablaLiquidos[Liquidos.Circuito_Liquido[10]].bAgitador);

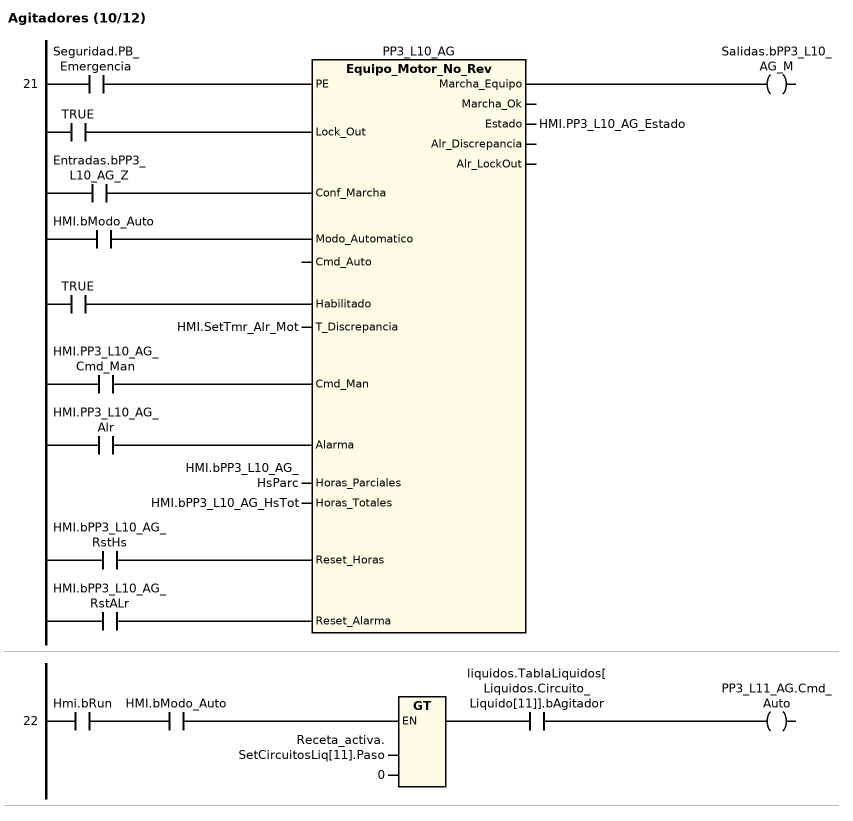
// NETWORK 21
PP3_L10_AG(
    PE := Seguridad.PB_Emergencia,
    Lock_Out := TRUE,
    Conf_Marcha := Entradas.bPP3_L10_AG_Z,
    Modo_Automatico := HMI.bModo_Auto,
    Habilitado := TRUE,
    T_Discrepancia := HMI.SetTmr_Alr_Mot,
    Cmd_Man := HMI.PP3_L10_AG_Cmd_Man,
    Alarma := HMI.PP3_L10_AG_Alr,
    Horas_Parciales := HMI.bPP3_L10_AG_HsParc,
    Horas_Totales := HMI.bPP3_L10_AG_HsTot,
    Reset_Horas := HMI.bPP3_L10_AG_RstHs,
    Reset_Alarma := HMI.bPP3_L10_AG_RstALr,
    Estado => HMI.PP3_L10_AG_Estado); // Equipo_Motor_No_Rev
Salidas.bPP3_L10_AG_M := PP3_L10_AG.Marcha_Equipo;

// NETWORK 22
PP3_L11_AG.Cmd_Auto := (Hmi.bRun AND HMI.bModo_Auto AND Receta_activa.SetCircuitosLiq[11].Paso > 0) AND (liquidos.TablaLiquidos[Liquidos.Circuito_Liquido[11]].bAgitador);

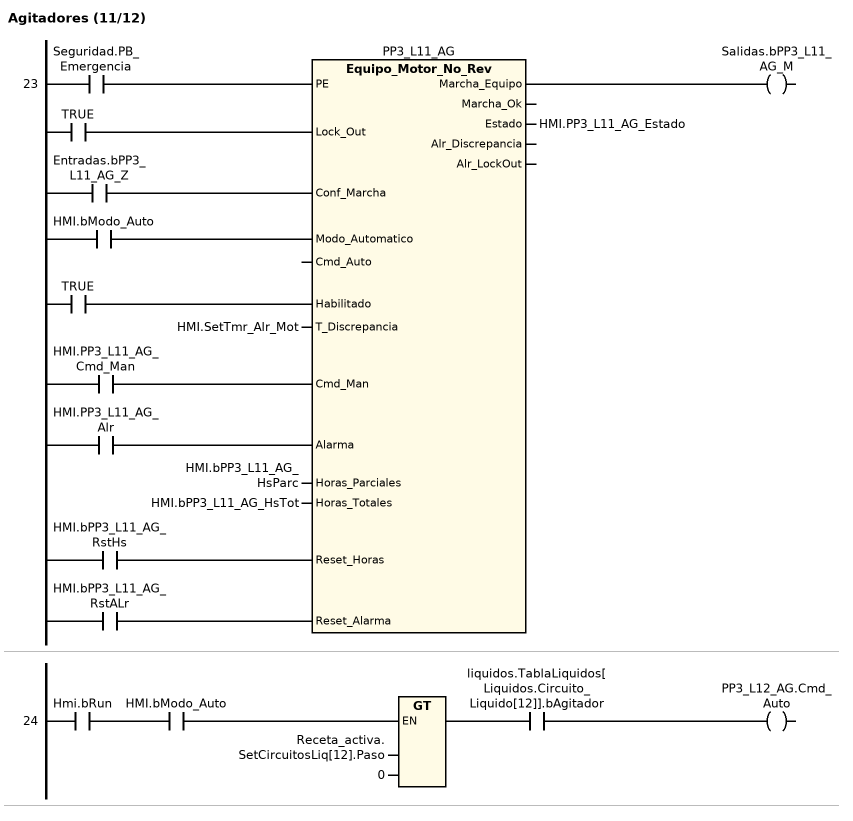
// NETWORK 23
PP3_L11_AG(
    PE := Seguridad.PB_Emergencia,
    Lock_Out := TRUE,
    Conf_Marcha := Entradas.bPP3_L11_AG_Z,
    Modo_Automatico := HMI.bModo_Auto,
    Habilitado := TRUE,
    T_Discrepancia := HMI.SetTmr_Alr_Mot,
    Cmd_Man := HMI.PP3_L11_AG_Cmd_Man,
    Alarma := HMI.PP3_L11_AG_Alr,
    Horas_Parciales := HMI.bPP3_L11_AG_HsParc,
    Horas_Totales := HMI.bPP3_L11_AG_HsTot,
    Reset_Horas := HMI.bPP3_L11_AG_RstHs,
    Reset_Alarma := HMI.bPP3_L11_AG_RstALr,
    Estado => HMI.PP3_L11_AG_Estado); // Equipo_Motor_No_Rev
Salidas.bPP3_L11_AG_M := PP3_L11_AG.Marcha_Equipo;

// NETWORK 24
PP3_L12_AG.Cmd_Auto := (Hmi.bRun AND HMI.bModo_Auto AND Receta_activa.SetCircuitosLiq[12].Paso > 0) AND (liquidos.TablaLiquidos[Liquidos.Circuito_Liquido[12]].bAgitador);

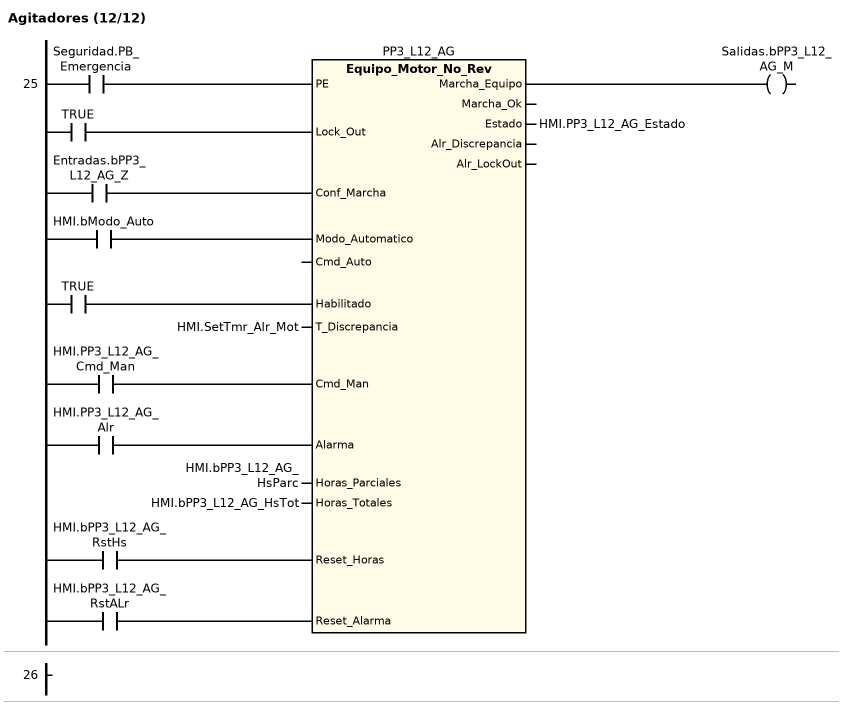
// NETWORK 25
PP3_L12_AG(
    PE := Seguridad.PB_Emergencia,
    Lock_Out := TRUE,
    Conf_Marcha := Entradas.bPP3_L12_AG_Z,
    Modo_Automatico := HMI.bModo_Auto,
    Habilitado := TRUE,
    T_Discrepancia := HMI.SetTmr_Alr_Mot,
    Cmd_Man := HMI.PP3_L12_AG_Cmd_Man,
    Alarma := HMI.PP3_L12_AG_Alr,
    Horas_Parciales := HMI.bPP3_L12_AG_HsParc,
    Horas_Totales := HMI.bPP3_L12_AG_HsTot,
    Reset_Horas := HMI.bPP3_L12_AG_RstHs,
    Reset_Alarma := HMI.bPP3_L12_AG_RstALr,
    Estado => HMI.PP3_L12_AG_Estado); // Equipo_Motor_No_Rev
Salidas.bPP3_L12_AG_M := PP3_L12_AG.Marcha_Equipo;

// NETWORK 26

END_PROGRAM

// ---- POUs/Puesto_Calibracion_1/Circuito_L1.TcPOU
PROGRAM Circuito_L1
VAR_INPUT
	Modo_Calibrar_L1: BOOL;
END_VAR

VAR
	fbLavado_L1 :LavadoCircuitoLiquidos;
	bhs :BOOL;
	rhs :REAL;
	ihs :INT;
	whs :WORD;
	ths :TIME;
	fbBomba_L1 :Equipo_Motor_ATV320;
	Totalizador_L1: Totalizador;
	Reset_TotL1:BOOL;
	ControlValv_ioLink_V1: ControlValv_ioLink;
	ControlValv_ioLink_V2: ControlValv_ioLink;
	ControlValv_ioLink_V3: ControlValv_ioLink;
	ControlValv_ioLink_V4: ControlValv_ioLink;
	Falla_L1_V1:BOOL;
	Falla_L1_V2:BOOL;
	Falla_L1_V3:BOOL;
	Falla_L1_V4:BOOL;
	Balanza_PU1_WT1: Balanza;
	dHS:DINT;
	TOF_calibradoIBC: TOF;
	TDemoraInyectar: TON;
	SetDemoraInyeccion: REAL;
	Volumen_L1: REAL;
	AuxVol: REAL;
	Total: REAL;
	auxIniCal: BOOL;
	Calculo_caudal_L1: Calculo_caudal;
	PID_L1_SP: REAL;
	PID_L1_PV: REAL;
	CorrecionCaudalxOffset_L1: CorrecionCaudalxOffset;
	tInyeccion: TON;
	PID_L1_manual: REAL;
	PID_L1: FB_PID;
	PID_L1_Kp: REAL := 0.1;
	PID_L1_Ti: REAL := 100;
	PID_L1_auto: BOOL;
	PID_L1_reset: BOOL;
	PID_L1_bMuerta: REAL := 5;
	Tiempo_seg_to_TIME_DemoraInyec: Tiempo_seg_to_TIME;
	AuxTDemoraInyec: TIME;
	Tiempo_TIME_to_seg_InyCal: Tiempo_TIME_to_seg;
	AuxInyCal:TIME;
	ProductoAsociado:STRING;
	Lavagem_Circuito01: Lavagem;
	RTRIG: ARRAY[1..10] OF R_TRIG;
	FiltroTeste: Filtro2;
END_VAR	
VAR PERSISTENT
	UltimaCalibracao	:UDINT;	//Data e hora da ultima calibração
END_VAR
VAR // added by the converter: edge detectors and wires of the graphical bodies
    _w1, _w2, _w3, _w4, _w5, _w6, _w7, _w8, _w9, _w10, _w11, _w12 : BOOL;
    _ft1 : F_TRIG;
    _rt1 : R_TRIG;
END_VAR

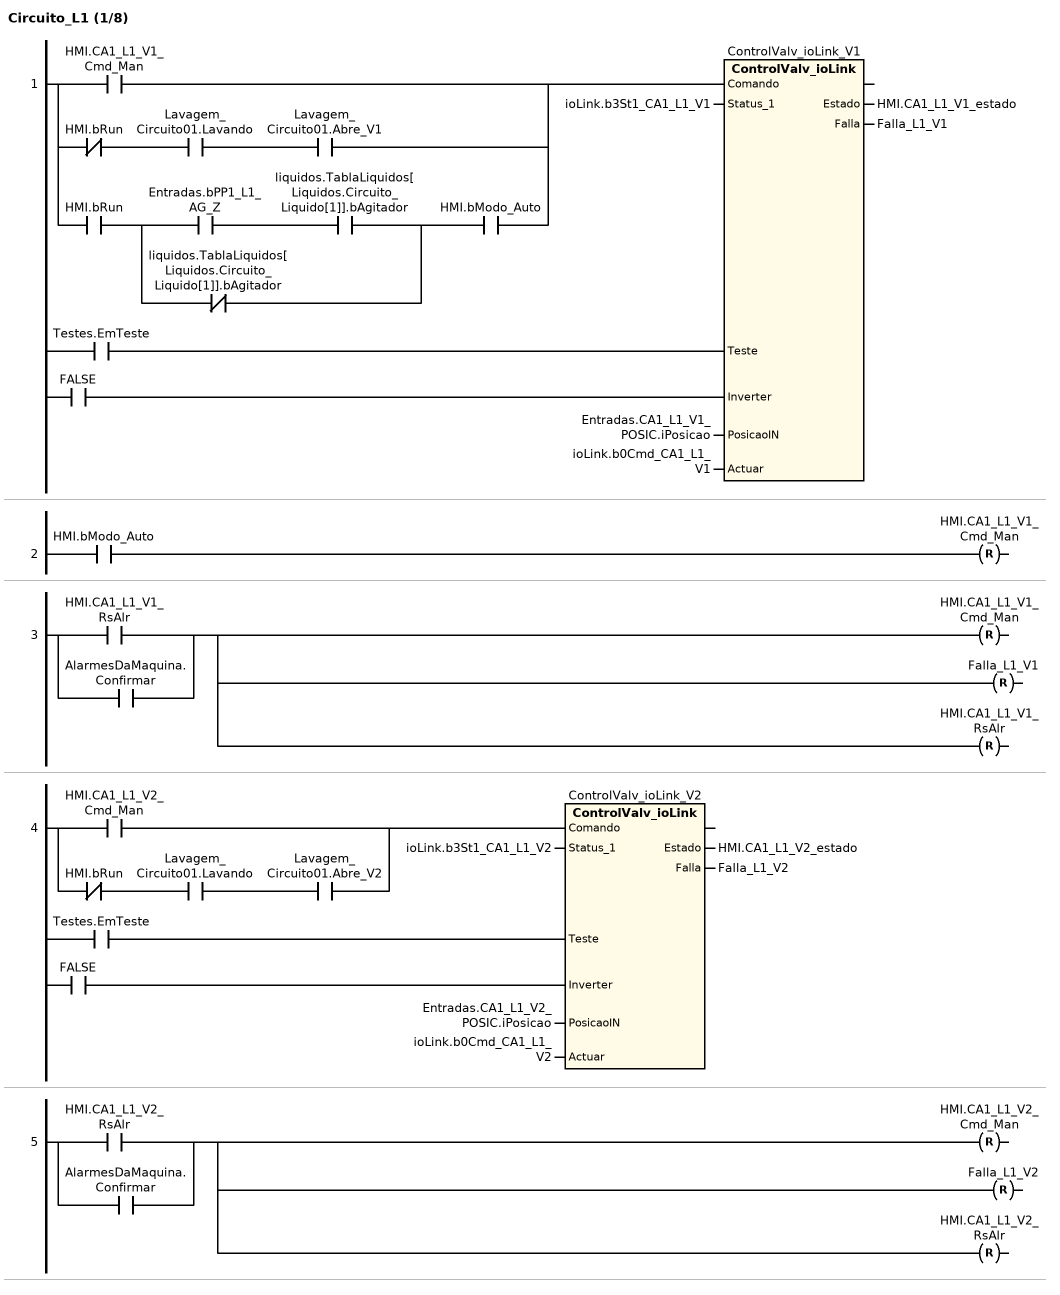
// NETWORK 1
ControlValv_ioLink_V1(
    Comando := HMI.CA1_L1_V1_Cmd_Man OR NOT HMI.bRun AND Lavagem_Circuito01.Lavando AND Lavagem_Circuito01.Abre_V1 OR HMI.bRun AND (Entradas.bPP1_L1_AG_Z AND (liquidos.TablaLiquidos[Liquidos.Circuito_Liquido[1]].bAgitador) OR NOT (liquidos.TablaLiquidos[Liquidos.Circuito_Liquido[1]].bAgitador)) AND HMI.bModo_Auto,
    Status_1 := ioLink.b3St1_CA1_L1_V1,
    Teste := Testes.EmTeste,
    Inverter := FALSE,
    PosicaoIN := Entradas.CA1_L1_V1_POSIC.iPosicao,
    Actuar := ioLink.b0Cmd_CA1_L1_V1,
    Estado => HMI.CA1_L1_V1_estado,
    Falla => Falla_L1_V1); // ControlValv_ioLink

// NETWORK 2
HMI.CA1_L1_V1_Cmd_Man R= HMI.bModo_Auto;

// NETWORK 3
_w1 := HMI.CA1_L1_V1_RsAlr OR AlarmesDaMaquina.Confirmar;
HMI.CA1_L1_V1_Cmd_Man R= _w1;
Falla_L1_V1 R= _w1;
HMI.CA1_L1_V1_RsAlr R= _w1;

// NETWORK 4
ControlValv_ioLink_V2(
    Comando := HMI.CA1_L1_V2_Cmd_Man OR NOT HMI.bRun AND Lavagem_Circuito01.Lavando AND Lavagem_Circuito01.Abre_V2,
    Status_1 := ioLink.b3St1_CA1_L1_V2,
    Teste := Testes.EmTeste,
    Inverter := FALSE,
    PosicaoIN := Entradas.CA1_L1_V2_POSIC.iPosicao,
    Actuar := ioLink.b0Cmd_CA1_L1_V2,
    Estado => HMI.CA1_L1_V2_estado,
    Falla => Falla_L1_V2); // ControlValv_ioLink

// NETWORK 5
_w2 := HMI.CA1_L1_V2_RsAlr OR AlarmesDaMaquina.Confirmar;
HMI.CA1_L1_V2_Cmd_Man R= _w2;
Falla_L1_V2 R= _w2;
HMI.CA1_L1_V2_RsAlr R= _w2;

